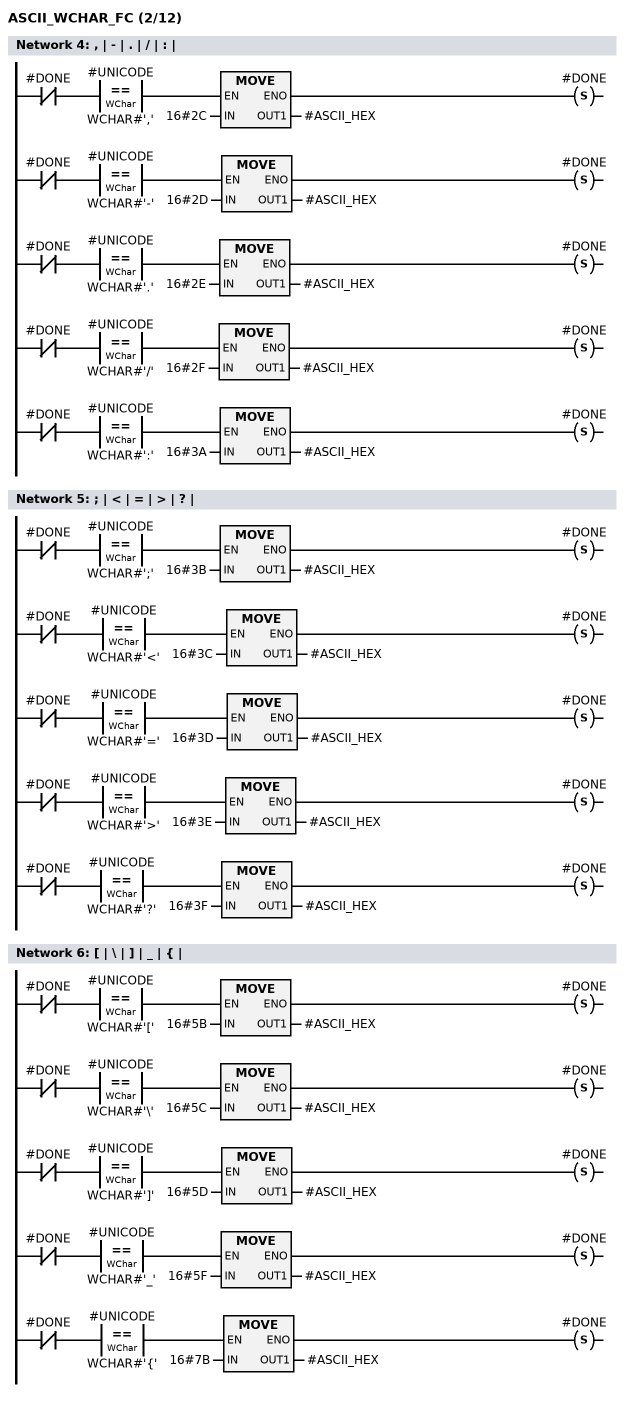
   RUNG wire#powerrail
      I_Contact( #DONE )
      { S7_Templates := "SrcType := WChar" } EQ_Contact(in1 := #UNICODE, in2 := WCHAR#',')
      Move(in := 16#2C, out1 => #ASCII_HEX)
      S_Coil( #DONE )
   END_RUNG
   RUNG wire#powerrail
      I_Contact( #DONE )
      { S7_Templates := "SrcType := WChar" } EQ_Contact(in1 := #UNICODE, in2 := WCHAR#'-')
      Move(in := 16#2D, out1 => #ASCII_HEX)
      S_Coil( #DONE )
   END_RUNG
   RUNG wire#powerrail
      I_Contact( #DONE )
      { S7_Templates := "SrcType := WChar" } EQ_Contact(in1 := #UNICODE, in2 := WCHAR#'.')
      Move(in := 16#2E, out1 => #ASCII_HEX)
      S_Coil( #DONE )
   END_RUNG
   RUNG wire#powerrail
      I_Contact( #DONE )
      { S7_Templates := "SrcType := WChar" } EQ_Contact(in1 := #UNICODE, in2 := WCHAR#'/')
      Move(in := 16#2F, out1 => #ASCII_HEX)
      S_Coil( #DONE )
   END_RUNG
   RUNG wire#powerrail
      I_Contact( #DONE )
      { S7_Templates := "SrcType := WChar" } EQ_Contact(in1 := #UNICODE, in2 := WCHAR#':')
      Move(in := 16#3A, out1 => #ASCII_HEX)
      S_Coil( #DONE )
   END_RUNG
   // the same network as SCL:
   IF NOT #DONE AND (#UNICODE = WCHAR#',') THEN
       #ASCII_HEX := 16#2C;
       #DONE := TRUE;
   END_IF;
   IF NOT #DONE AND (#UNICODE = WCHAR#'-') THEN
       #ASCII_HEX := 16#2D;
       #DONE := TRUE;
   END_IF;
   IF NOT #DONE AND (#UNICODE = WCHAR#'.') THEN
       #ASCII_HEX := 16#2E;
       #DONE := TRUE;
   END_IF;
   IF NOT #DONE AND (#UNICODE = WCHAR#'/') THEN
       #ASCII_HEX := 16#2F;
       #DONE := TRUE;
   END_IF;
   IF NOT #DONE AND (#UNICODE = WCHAR#':') THEN
       #ASCII_HEX := 16#3A;
       #DONE := TRUE;
   END_IF;
END_REGION

REGION Network 5: ; | < | = | > | ? |
   RUNG wire#powerrail
      I_Contact( #DONE )
      { S7_Templates := "SrcType := WChar" } EQ_Contact(in1 := #UNICODE, in2 := WCHAR#';')
      Move(in := 16#3B, out1 => #ASCII_HEX)
      S_Coil( #DONE )
   END_RUNG
   RUNG wire#powerrail
      I_Contact( #DONE )
      { S7_Templates := "SrcType := WChar" } EQ_Contact(in1 := #UNICODE, in2 := WCHAR#'<')
      Move(in := 16#3C, out1 => #ASCII_HEX)
      S_Coil( #DONE )
   END_RUNG
   RUNG wire#powerrail
      I_Contact( #DONE )
      { S7_Templates := "SrcType := WChar" } EQ_Contact(in1 := #UNICODE, in2 := WCHAR#'=')
      Move(in := 16#3D, out1 => #ASCII_HEX)
      S_Coil( #DONE )
   END_RUNG
   RUNG wire#powerrail
      I_Contact( #DONE )
      { S7_Templates := "SrcType := WChar" } EQ_Contact(in1 := #UNICODE, in2 := WCHAR#'>')
      Move(in := 16#3E, out1 => #ASCII_HEX)
      S_Coil( #DONE )
   END_RUNG
   RUNG wire#powerrail
      I_Contact( #DONE )
      { S7_Templates := "SrcType := WChar" } EQ_Contact(in1 := #UNICODE, in2 := WCHAR#'?')
      Move(in := 16#3F, out1 => #ASCII_HEX)
      S_Coil( #DONE )
   END_RUNG
   // the same network as SCL:
   IF NOT #DONE AND (#UNICODE = WCHAR#';') THEN
       #ASCII_HEX := 16#3B;
       #DONE := TRUE;
   END_IF;
   IF NOT #DONE AND (#UNICODE = WCHAR#'<') THEN
       #ASCII_HEX := 16#3C;
       #DONE := TRUE;
   END_IF;
   IF NOT #DONE AND (#UNICODE = WCHAR#'=') THEN
       #ASCII_HEX := 16#3D;
       #DONE := TRUE;
   END_IF;
   IF NOT #DONE AND (#UNICODE = WCHAR#'>') THEN
       #ASCII_HEX := 16#3E;
       #DONE := TRUE;
   END_IF;
   IF NOT #DONE AND (#UNICODE = WCHAR#'?') THEN
       #ASCII_HEX := 16#3F;
       #DONE := TRUE;
   END_IF;
END_REGION

REGION Network 6: [ | \ | ] | _ | { |
   RUNG wire#powerrail
      I_Contact( #DONE )
      { S7_Templates := "SrcType := WChar" } EQ_Contact(in1 := #UNICODE, in2 := WCHAR#'[')
      Move(in := 16#5B, out1 => #ASCII_HEX)
      S_Coil( #DONE )
   END_RUNG
   RUNG wire#powerrail
      I_Contact( #DONE )
      { S7_Templates := "SrcType := WChar" } EQ_Contact(in1 := #UNICODE, in2 := WCHAR#'\')
      Move(in := 16#5C, out1 => #ASCII_HEX)
      S_Coil( #DONE )
   END_RUNG
   RUNG wire#powerrail
      I_Contact( #DONE )
      { S7_Templates := "SrcType := WChar" } EQ_Contact(in1 := #UNICODE, in2 := WCHAR#']')
      Move(in := 16#5D, out1 => #ASCII_HEX)
      S_Coil( #DONE )
   END_RUNG
   RUNG wire#powerrail
      I_Contact( #DONE )
      { S7_Templates := "SrcType := WChar" } EQ_Contact(in1 := #UNICODE, in2 := WCHAR#'_')
      Move(in := 16#5F, out1 => #ASCII_HEX)
      S_Coil( #DONE )
   END_RUNG
   RUNG wire#powerrail
      I_Contact( #DONE )
      { S7_Templates := "SrcType := WChar" } EQ_Contact(in1 := #UNICODE, in2 := WCHAR#'{')
      Move(in := 16#7B, out1 => #ASCII_HEX)
      S_Coil( #DONE )
   END_RUNG
   // the same network as SCL:
   IF NOT #DONE AND (#UNICODE = WCHAR#'[') THEN
       #ASCII_HEX := 16#5B;
       #DONE := TRUE;
   END_IF;
   IF NOT #DONE AND (#UNICODE = WCHAR#'\') THEN
       #ASCII_HEX := 16#5C;
       #DONE := TRUE;
   END_IF;
   IF NOT #DONE AND (#UNICODE = WCHAR#']') THEN
       #ASCII_HEX := 16#5D;
       #DONE := TRUE;
   END_IF;
   IF NOT #DONE AND (#UNICODE = WCHAR#'_') THEN
       #ASCII_HEX := 16#5F;
       #DONE := TRUE;
   END_IF;
   IF NOT #DONE AND (#UNICODE = WCHAR#'{') THEN
       #ASCII_HEX := 16#7B;
       #DONE := TRUE;
   END_IF;
END_REGION

REGION Network 7: } | | |
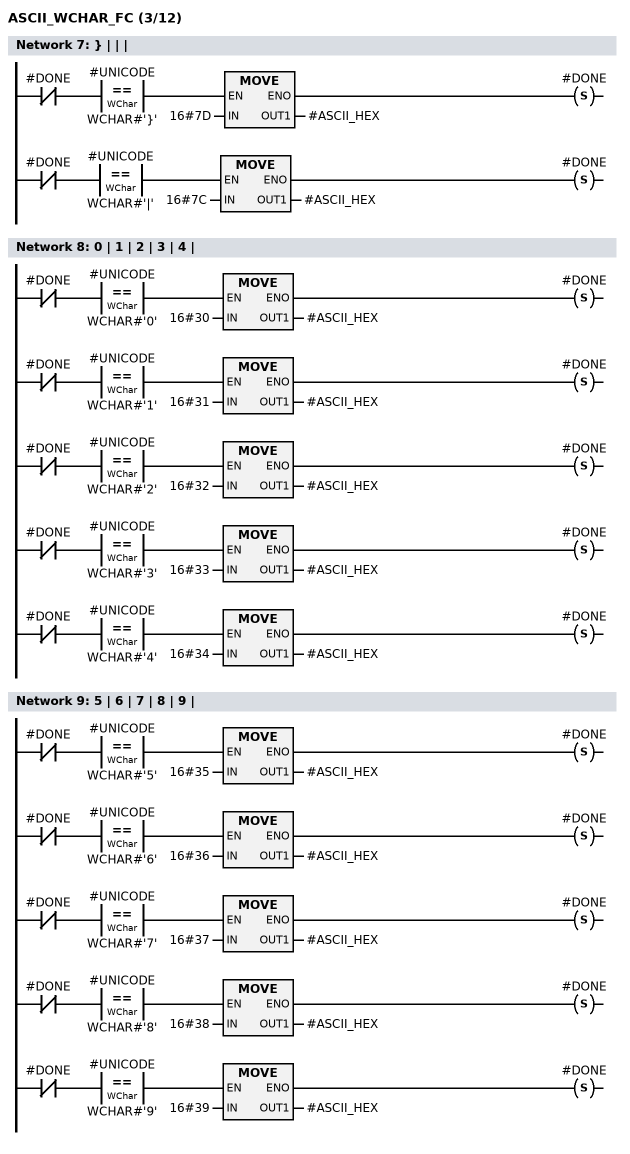
   RUNG wire#powerrail
      I_Contact( #DONE )
      { S7_Templates := "SrcType := WChar" } EQ_Contact(in1 := #UNICODE, in2 := WCHAR#'}')
      Move(in := 16#7D, out1 => #ASCII_HEX)
      S_Coil( #DONE )
   END_RUNG
   RUNG wire#powerrail
      I_Contact( #DONE )
      { S7_Templates := "SrcType := WChar" } EQ_Contact(in1 := #UNICODE, in2 := WCHAR#'|')
      Move(in := 16#7C, out1 => #ASCII_HEX)
      S_Coil( #DONE )
   END_RUNG
   // the same network as SCL:
   IF NOT #DONE AND (#UNICODE = WCHAR#'}') THEN
       #ASCII_HEX := 16#7D;
       #DONE := TRUE;
   END_IF;
   IF NOT #DONE AND (#UNICODE = WCHAR#'|') THEN
       #ASCII_HEX := 16#7C;
       #DONE := TRUE;
   END_IF;
END_REGION

REGION Network 8: 0 | 1 | 2 | 3 | 4 |
   RUNG wire#powerrail
      I_Contact( #DONE )
      { S7_Templates := "SrcType := WChar" } EQ_Contact(in1 := #UNICODE, in2 := WCHAR#'0')
      Move(in := 16#30, out1 => #ASCII_HEX)
      S_Coil( #DONE )
   END_RUNG
   RUNG wire#powerrail
      I_Contact( #DONE )
      { S7_Templates := "SrcType := WChar" } EQ_Contact(in1 := #UNICODE, in2 := WCHAR#'1')
      Move(in := 16#31, out1 => #ASCII_HEX)
      S_Coil( #DONE )
   END_RUNG
   RUNG wire#powerrail
      I_Contact( #DONE )
      { S7_Templates := "SrcType := WChar" } EQ_Contact(in1 := #UNICODE, in2 := WCHAR#'2')
      Move(in := 16#32, out1 => #ASCII_HEX)
      S_Coil( #DONE )
   END_RUNG
   RUNG wire#powerrail
      I_Contact( #DONE )
      { S7_Templates := "SrcType := WChar" } EQ_Contact(in1 := #UNICODE, in2 := WCHAR#'3')
      Move(in := 16#33, out1 => #ASCII_HEX)
      S_Coil( #DONE )
   END_RUNG
   RUNG wire#powerrail
      I_Contact( #DONE )
      { S7_Templates := "SrcType := WChar" } EQ_Contact(in1 := #UNICODE, in2 := WCHAR#'4')
      Move(in := 16#34, out1 => #ASCII_HEX)
      S_Coil( #DONE )
   END_RUNG
   // the same network as SCL:
   IF NOT #DONE AND (#UNICODE = WCHAR#'0') THEN
       #ASCII_HEX := 16#30;
       #DONE := TRUE;
   END_IF;
   IF NOT #DONE AND (#UNICODE = WCHAR#'1') THEN
       #ASCII_HEX := 16#31;
       #DONE := TRUE;
   END_IF;
   IF NOT #DONE AND (#UNICODE = WCHAR#'2') THEN
       #ASCII_HEX := 16#32;
       #DONE := TRUE;
   END_IF;
   IF NOT #DONE AND (#UNICODE = WCHAR#'3') THEN
       #ASCII_HEX := 16#33;
       #DONE := TRUE;
   END_IF;
   IF NOT #DONE AND (#UNICODE = WCHAR#'4') THEN
       #ASCII_HEX := 16#34;
       #DONE := TRUE;
   END_IF;
END_REGION

REGION Network 9: 5 | 6 | 7 | 8 | 9 |
   RUNG wire#powerrail
      I_Contact( #DONE )
      { S7_Templates := "SrcType := WChar" } EQ_Contact(in1 := #UNICODE, in2 := WCHAR#'5')
      Move(in := 16#35, out1 => #ASCII_HEX)
      S_Coil( #DONE )
   END_RUNG
   RUNG wire#powerrail
      I_Contact( #DONE )
      { S7_Templates := "SrcType := WChar" } EQ_Contact(in1 := #UNICODE, in2 := WCHAR#'6')
      Move(in := 16#36, out1 => #ASCII_HEX)
      S_Coil( #DONE )
   END_RUNG
   RUNG wire#powerrail
      I_Contact( #DONE )
      { S7_Templates := "SrcType := WChar" } EQ_Contact(in1 := #UNICODE, in2 := WCHAR#'7')
      Move(in := 16#37, out1 => #ASCII_HEX)
      S_Coil( #DONE )
   END_RUNG
   RUNG wire#powerrail
      I_Contact( #DONE )
      { S7_Templates := "SrcType := WChar" } EQ_Contact(in1 := #UNICODE, in2 := WCHAR#'8')
      Move(in := 16#38, out1 => #ASCII_HEX)
      S_Coil( #DONE )
   END_RUNG
   RUNG wire#powerrail
      I_Contact( #DONE )
      { S7_Templates := "SrcType := WChar" } EQ_Contact(in1 := #UNICODE, in2 := WCHAR#'9')
      Move(in := 16#39, out1 => #ASCII_HEX)
      S_Coil( #DONE )
   END_RUNG
   // the same network as SCL:
   IF NOT #DONE AND (#UNICODE = WCHAR#'5') THEN
       #ASCII_HEX := 16#35;
       #DONE := TRUE;
   END_IF;
   IF NOT #DONE AND (#UNICODE = WCHAR#'6') THEN
       #ASCII_HEX := 16#36;
       #DONE := TRUE;
   END_IF;
   IF NOT #DONE AND (#UNICODE = WCHAR#'7') THEN
       #ASCII_HEX := 16#37;
       #DONE := TRUE;
   END_IF;
   IF NOT #DONE AND (#UNICODE = WCHAR#'8') THEN
       #ASCII_HEX := 16#38;
       #DONE := TRUE;
   END_IF;
   IF NOT #DONE AND (#UNICODE = WCHAR#'9') THEN
       #ASCII_HEX := 16#39;
       #DONE := TRUE;
   END_IF;
END_REGION

REGION Network 10: А | Б | В | Г | Д |
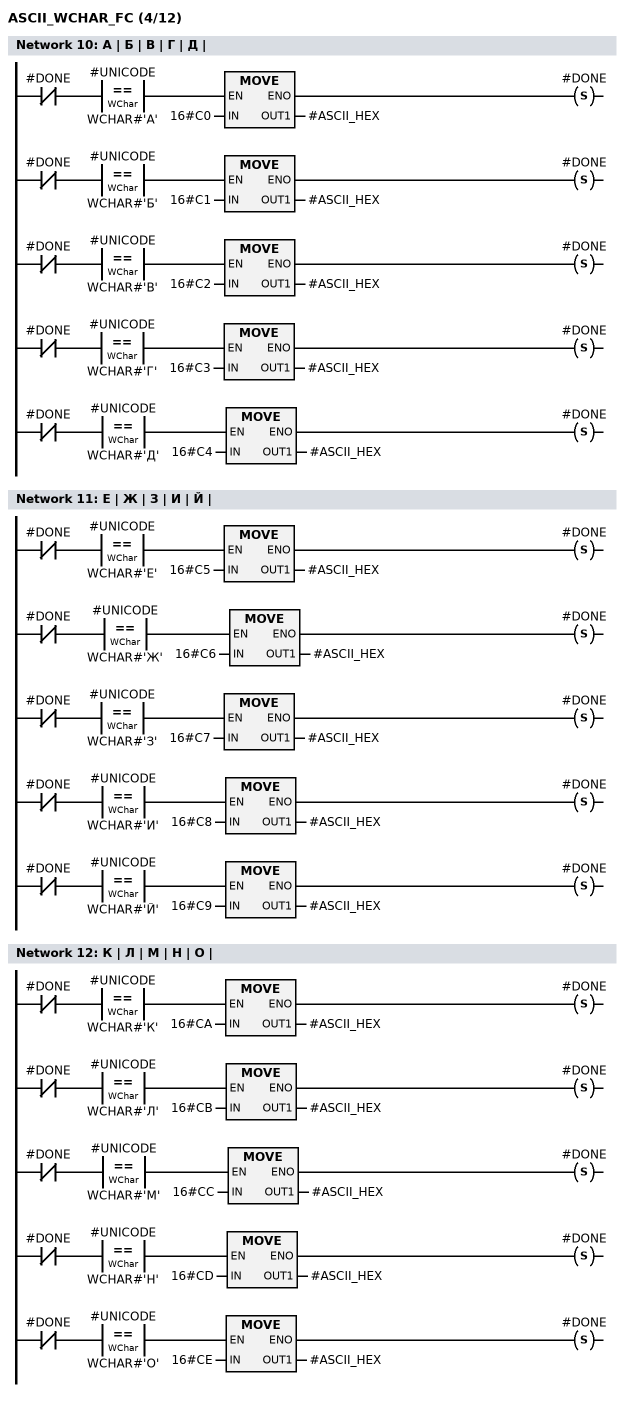
   RUNG wire#powerrail
      I_Contact( #DONE )
      { S7_Templates := "SrcType := WChar" } EQ_Contact(in1 := #UNICODE, in2 := WCHAR#'А')
      Move(in := 16#C0, out1 => #ASCII_HEX)
      S_Coil( #DONE )
   END_RUNG
   RUNG wire#powerrail
      I_Contact( #DONE )
      { S7_Templates := "SrcType := WChar" } EQ_Contact(in1 := #UNICODE, in2 := WCHAR#'Б')
      Move(in := 16#C1, out1 => #ASCII_HEX)
      S_Coil( #DONE )
   END_RUNG
   RUNG wire#powerrail
      I_Contact( #DONE )
      { S7_Templates := "SrcType := WChar" } EQ_Contact(in1 := #UNICODE, in2 := WCHAR#'В')
      Move(in := 16#C2, out1 => #ASCII_HEX)
      S_Coil( #DONE )
   END_RUNG
   RUNG wire#powerrail
      I_Contact( #DONE )
      { S7_Templates := "SrcType := WChar" } EQ_Contact(in1 := #UNICODE, in2 := WCHAR#'Г')
      Move(in := 16#C3, out1 => #ASCII_HEX)
      S_Coil( #DONE )
   END_RUNG
   RUNG wire#powerrail
      I_Contact( #DONE )
      { S7_Templates := "SrcType := WChar" } EQ_Contact(in1 := #UNICODE, in2 := WCHAR#'Д')
      Move(in := 16#C4, out1 => #ASCII_HEX)
      S_Coil( #DONE )
   END_RUNG
   // the same network as SCL:
   IF NOT #DONE AND (#UNICODE = WCHAR#'А') THEN
       #ASCII_HEX := 16#C0;
       #DONE := TRUE;
   END_IF;
   IF NOT #DONE AND (#UNICODE = WCHAR#'Б') THEN
       #ASCII_HEX := 16#C1;
       #DONE := TRUE;
   END_IF;
   IF NOT #DONE AND (#UNICODE = WCHAR#'В') THEN
       #ASCII_HEX := 16#C2;
       #DONE := TRUE;
   END_IF;
   IF NOT #DONE AND (#UNICODE = WCHAR#'Г') THEN
       #ASCII_HEX := 16#C3;
       #DONE := TRUE;
   END_IF;
   IF NOT #DONE AND (#UNICODE = WCHAR#'Д') THEN
       #ASCII_HEX := 16#C4;
       #DONE := TRUE;
   END_IF;
END_REGION

REGION Network 11: Е | Ж | З | И | Й |
   RUNG wire#powerrail
      I_Contact( #DONE )
      { S7_Templates := "SrcType := WChar" } EQ_Contact(in1 := #UNICODE, in2 := WCHAR#'Е')
      Move(in := 16#C5, out1 => #ASCII_HEX)
      S_Coil( #DONE )
   END_RUNG
   RUNG wire#powerrail
      I_Contact( #DONE )
      { S7_Templates := "SrcType := WChar" } EQ_Contact(in1 := #UNICODE, in2 := WCHAR#'Ж')
      Move(in := 16#C6, out1 => #ASCII_HEX)
      S_Coil( #DONE )
   END_RUNG
   RUNG wire#powerrail
      I_Contact( #DONE )
      { S7_Templates := "SrcType := WChar" } EQ_Contact(in1 := #UNICODE, in2 := WCHAR#'З')
      Move(in := 16#C7, out1 => #ASCII_HEX)
      S_Coil( #DONE )
   END_RUNG
   RUNG wire#powerrail
      I_Contact( #DONE )
      { S7_Templates := "SrcType := WChar" } EQ_Contact(in1 := #UNICODE, in2 := WCHAR#'И')
      Move(in := 16#C8, out1 => #ASCII_HEX)
      S_Coil( #DONE )
   END_RUNG
   RUNG wire#powerrail
      I_Contact( #DONE )
      { S7_Templates := "SrcType := WChar" } EQ_Contact(in1 := #UNICODE, in2 := WCHAR#'Й')
      Move(in := 16#C9, out1 => #ASCII_HEX)
      S_Coil( #DONE )
   END_RUNG
   // the same network as SCL:
   IF NOT #DONE AND (#UNICODE = WCHAR#'Е') THEN
       #ASCII_HEX := 16#C5;
       #DONE := TRUE;
   END_IF;
   IF NOT #DONE AND (#UNICODE = WCHAR#'Ж') THEN
       #ASCII_HEX := 16#C6;
       #DONE := TRUE;
   END_IF;
   IF NOT #DONE AND (#UNICODE = WCHAR#'З') THEN
       #ASCII_HEX := 16#C7;
       #DONE := TRUE;
   END_IF;
   IF NOT #DONE AND (#UNICODE = WCHAR#'И') THEN
       #ASCII_HEX := 16#C8;
       #DONE := TRUE;
   END_IF;
   IF NOT #DONE AND (#UNICODE = WCHAR#'Й') THEN
       #ASCII_HEX := 16#C9;
       #DONE := TRUE;
   END_IF;
END_REGION

REGION Network 12: К | Л | М | Н | О |
   RUNG wire#powerrail
      I_Contact( #DONE )
      { S7_Templates := "SrcType := WChar" } EQ_Contact(in1 := #UNICODE, in2 := WCHAR#'К')
      Move(in := 16#CA, out1 => #ASCII_HEX)
      S_Coil( #DONE )
   END_RUNG
   RUNG wire#powerrail
      I_Contact( #DONE )
      { S7_Templates := "SrcType := WChar" } EQ_Contact(in1 := #UNICODE, in2 := WCHAR#'Л')
      Move(in := 16#CB, out1 => #ASCII_HEX)
      S_Coil( #DONE )
   END_RUNG
   RUNG wire#powerrail
      I_Contact( #DONE )
      { S7_Templates := "SrcType := WChar" } EQ_Contact(in1 := #UNICODE, in2 := WCHAR#'М')
      Move(in := 16#CC, out1 => #ASCII_HEX)
      S_Coil( #DONE )
   END_RUNG
   RUNG wire#powerrail
      I_Contact( #DONE )
      { S7_Templates := "SrcType := WChar" } EQ_Contact(in1 := #UNICODE, in2 := WCHAR#'Н')
      Move(in := 16#CD, out1 => #ASCII_HEX)
      S_Coil( #DONE )
   END_RUNG
   RUNG wire#powerrail
      I_Contact( #DONE )
      { S7_Templates := "SrcType := WChar" } EQ_Contact(in1 := #UNICODE, in2 := WCHAR#'О')
      Move(in := 16#CE, out1 => #ASCII_HEX)
      S_Coil( #DONE )
   END_RUNG
   // the same network as SCL:
   IF NOT #DONE AND (#UNICODE = WCHAR#'К') THEN
       #ASCII_HEX := 16#CA;
       #DONE := TRUE;
   END_IF;
   IF NOT #DONE AND (#UNICODE = WCHAR#'Л') THEN
       #ASCII_HEX := 16#CB;
       #DONE := TRUE;
   END_IF;
   IF NOT #DONE AND (#UNICODE = WCHAR#'М') THEN
       #ASCII_HEX := 16#CC;
       #DONE := TRUE;
   END_IF;
   IF NOT #DONE AND (#UNICODE = WCHAR#'Н') THEN
       #ASCII_HEX := 16#CD;
       #DONE := TRUE;
   END_IF;
   IF NOT #DONE AND (#UNICODE = WCHAR#'О') THEN
       #ASCII_HEX := 16#CE;
       #DONE := TRUE;
   END_IF;
END_REGION

REGION Network 13: П | Р | С | Т | У |
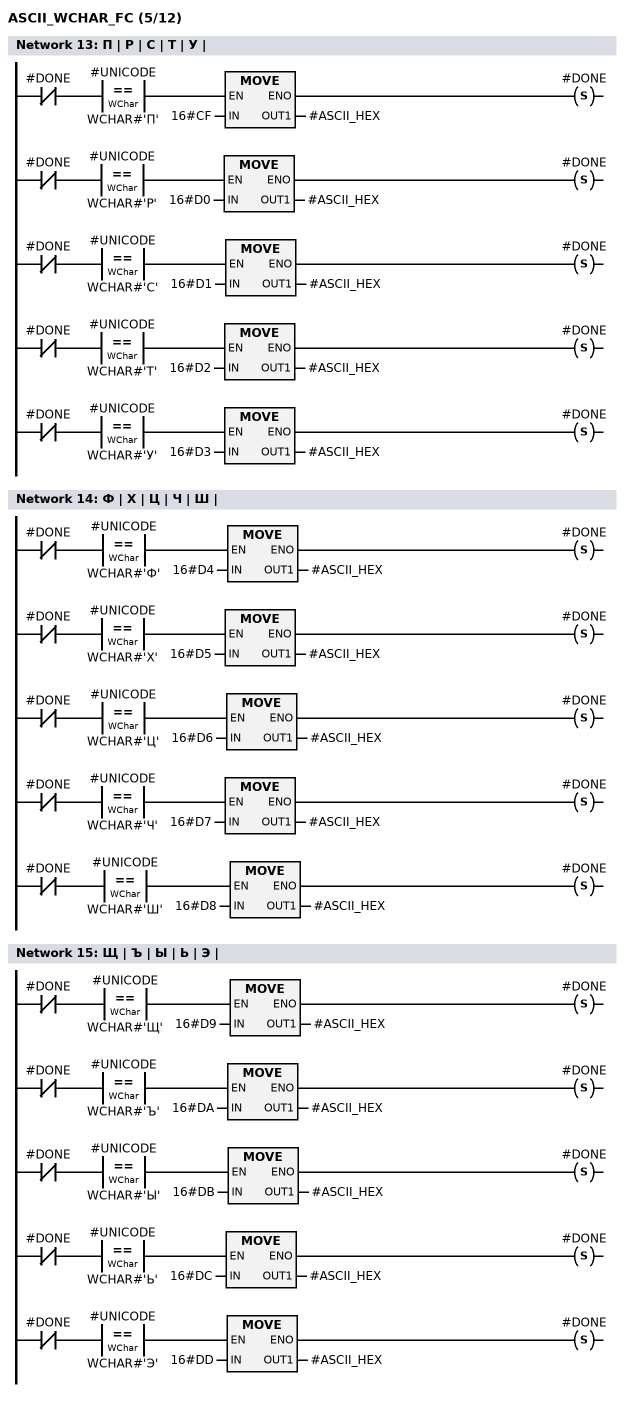
   RUNG wire#powerrail
      I_Contact( #DONE )
      { S7_Templates := "SrcType := WChar" } EQ_Contact(in1 := #UNICODE, in2 := WCHAR#'П')
      Move(in := 16#CF, out1 => #ASCII_HEX)
      S_Coil( #DONE )
   END_RUNG
   RUNG wire#powerrail
      I_Contact( #DONE )
      { S7_Templates := "SrcType := WChar" } EQ_Contact(in1 := #UNICODE, in2 := WCHAR#'Р')
      Move(in := 16#D0, out1 => #ASCII_HEX)
      S_Coil( #DONE )
   END_RUNG
   RUNG wire#powerrail
      I_Contact( #DONE )
      { S7_Templates := "SrcType := WChar" } EQ_Contact(in1 := #UNICODE, in2 := WCHAR#'С')
      Move(in := 16#D1, out1 => #ASCII_HEX)
      S_Coil( #DONE )
   END_RUNG
   RUNG wire#powerrail
      I_Contact( #DONE )
      { S7_Templates := "SrcType := WChar" } EQ_Contact(in1 := #UNICODE, in2 := WCHAR#'Т')
      Move(in := 16#D2, out1 => #ASCII_HEX)
      S_Coil( #DONE )
   END_RUNG
   RUNG wire#powerrail
      I_Contact( #DONE )
      { S7_Templates := "SrcType := WChar" } EQ_Contact(in1 := #UNICODE, in2 := WCHAR#'У')
      Move(in := 16#D3, out1 => #ASCII_HEX)
      S_Coil( #DONE )
   END_RUNG
   // the same network as SCL:
   IF NOT #DONE AND (#UNICODE = WCHAR#'П') THEN
       #ASCII_HEX := 16#CF;
       #DONE := TRUE;
   END_IF;
   IF NOT #DONE AND (#UNICODE = WCHAR#'Р') THEN
       #ASCII_HEX := 16#D0;
       #DONE := TRUE;
   END_IF;
   IF NOT #DONE AND (#UNICODE = WCHAR#'С') THEN
       #ASCII_HEX := 16#D1;
       #DONE := TRUE;
   END_IF;
   IF NOT #DONE AND (#UNICODE = WCHAR#'Т') THEN
       #ASCII_HEX := 16#D2;
       #DONE := TRUE;
   END_IF;
   IF NOT #DONE AND (#UNICODE = WCHAR#'У') THEN
       #ASCII_HEX := 16#D3;
       #DONE := TRUE;
   END_IF;
END_REGION

REGION Network 14: Ф | Х | Ц | Ч | Ш |
   RUNG wire#powerrail
      I_Contact( #DONE )
      { S7_Templates := "SrcType := WChar" } EQ_Contact(in1 := #UNICODE, in2 := WCHAR#'Ф')
      Move(in := 16#D4, out1 => #ASCII_HEX)
      S_Coil( #DONE )
   END_RUNG
   RUNG wire#powerrail
      I_Contact( #DONE )
      { S7_Templates := "SrcType := WChar" } EQ_Contact(in1 := #UNICODE, in2 := WCHAR#'Х')
      Move(in := 16#D5, out1 => #ASCII_HEX)
      S_Coil( #DONE )
   END_RUNG
   RUNG wire#powerrail
      I_Contact( #DONE )
      { S7_Templates := "SrcType := WChar" } EQ_Contact(in1 := #UNICODE, in2 := WCHAR#'Ц')
      Move(in := 16#D6, out1 => #ASCII_HEX)
      S_Coil( #DONE )
   END_RUNG
   RUNG wire#powerrail
      I_Contact( #DONE )
      { S7_Templates := "SrcType := WChar" } EQ_Contact(in1 := #UNICODE, in2 := WCHAR#'Ч')
      Move(in := 16#D7, out1 => #ASCII_HEX)
      S_Coil( #DONE )
   END_RUNG
   RUNG wire#powerrail
      I_Contact( #DONE )
      { S7_Templates := "SrcType := WChar" } EQ_Contact(in1 := #UNICODE, in2 := WCHAR#'Ш')
      Move(in := 16#D8, out1 => #ASCII_HEX)
      S_Coil( #DONE )
   END_RUNG
   // the same network as SCL:
   IF NOT #DONE AND (#UNICODE = WCHAR#'Ф') THEN
       #ASCII_HEX := 16#D4;
       #DONE := TRUE;
   END_IF;
   IF NOT #DONE AND (#UNICODE = WCHAR#'Х') THEN
       #ASCII_HEX := 16#D5;
       #DONE := TRUE;
   END_IF;
   IF NOT #DONE AND (#UNICODE = WCHAR#'Ц') THEN
       #ASCII_HEX := 16#D6;
       #DONE := TRUE;
   END_IF;
   IF NOT #DONE AND (#UNICODE = WCHAR#'Ч') THEN
       #ASCII_HEX := 16#D7;
       #DONE := TRUE;
   END_IF;
   IF NOT #DONE AND (#UNICODE = WCHAR#'Ш') THEN
       #ASCII_HEX := 16#D8;
       #DONE := TRUE;
   END_IF;
END_REGION

REGION Network 15: Щ | Ъ | Ы | Ь | Э |
   RUNG wire#powerrail
      I_Contact( #DONE )
      { S7_Templates := "SrcType := WChar" } EQ_Contact(in1 := #UNICODE, in2 := WCHAR#'Щ')
      Move(in := 16#D9, out1 => #ASCII_HEX)
      S_Coil( #DONE )
   END_RUNG
   RUNG wire#powerrail
      I_Contact( #DONE )
      { S7_Templates := "SrcType := WChar" } EQ_Contact(in1 := #UNICODE, in2 := WCHAR#'Ъ')
      Move(in := 16#DA, out1 => #ASCII_HEX)
      S_Coil( #DONE )
   END_RUNG
   RUNG wire#powerrail
      I_Contact( #DONE )
      { S7_Templates := "SrcType := WChar" } EQ_Contact(in1 := #UNICODE, in2 := WCHAR#'Ы')
      Move(in := 16#DB, out1 => #ASCII_HEX)
      S_Coil( #DONE )
   END_RUNG
   RUNG wire#powerrail
      I_Contact( #DONE )
      { S7_Templates := "SrcType := WChar" } EQ_Contact(in1 := #UNICODE, in2 := WCHAR#'Ь')
      Move(in := 16#DC, out1 => #ASCII_HEX)
      S_Coil( #DONE )
   END_RUNG
   RUNG wire#powerrail
      I_Contact( #DONE )
      { S7_Templates := "SrcType := WChar" } EQ_Contact(in1 := #UNICODE, in2 := WCHAR#'Э')
      Move(in := 16#DD, out1 => #ASCII_HEX)
      S_Coil( #DONE )
   END_RUNG
   // the same network as SCL:
   IF NOT #DONE AND (#UNICODE = WCHAR#'Щ') THEN
       #ASCII_HEX := 16#D9;
       #DONE := TRUE;
   END_IF;
   IF NOT #DONE AND (#UNICODE = WCHAR#'Ъ') THEN
       #ASCII_HEX := 16#DA;
       #DONE := TRUE;
   END_IF;
   IF NOT #DONE AND (#UNICODE = WCHAR#'Ы') THEN
       #ASCII_HEX := 16#DB;
       #DONE := TRUE;
   END_IF;
   IF NOT #DONE AND (#UNICODE = WCHAR#'Ь') THEN
       #ASCII_HEX := 16#DC;
       #DONE := TRUE;
   END_IF;
   IF NOT #DONE AND (#UNICODE = WCHAR#'Э') THEN
       #ASCII_HEX := 16#DD;
       #DONE := TRUE;
   END_IF;
END_REGION

REGION Network 16: Ю | Я |
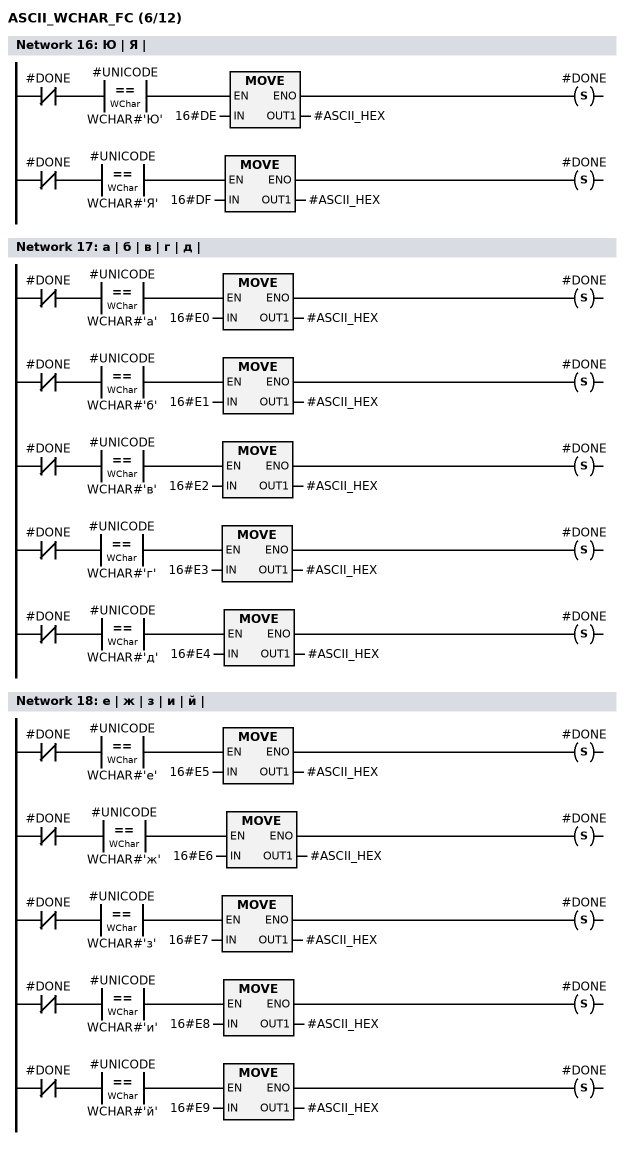
   RUNG wire#powerrail
      I_Contact( #DONE )
      { S7_Templates := "SrcType := WChar" } EQ_Contact(in1 := #UNICODE, in2 := WCHAR#'Ю')
      Move(in := 16#DE, out1 => #ASCII_HEX)
      S_Coil( #DONE )
   END_RUNG
   RUNG wire#powerrail
      I_Contact( #DONE )
      { S7_Templates := "SrcType := WChar" } EQ_Contact(in1 := #UNICODE, in2 := WCHAR#'Я')
      Move(in := 16#DF, out1 => #ASCII_HEX)
      S_Coil( #DONE )
   END_RUNG
   // the same network as SCL:
   IF NOT #DONE AND (#UNICODE = WCHAR#'Ю') THEN
       #ASCII_HEX := 16#DE;
       #DONE := TRUE;
   END_IF;
   IF NOT #DONE AND (#UNICODE = WCHAR#'Я') THEN
       #ASCII_HEX := 16#DF;
       #DONE := TRUE;
   END_IF;
END_REGION

REGION Network 17: а | б | в | г | д |
   RUNG wire#powerrail
      I_Contact( #DONE )
      { S7_Templates := "SrcType := WChar" } EQ_Contact(in1 := #UNICODE, in2 := WCHAR#'а')
      Move(in := 16#E0, out1 => #ASCII_HEX)
      S_Coil( #DONE )
   END_RUNG
   RUNG wire#powerrail
      I_Contact( #DONE )
      { S7_Templates := "SrcType := WChar" } EQ_Contact(in1 := #UNICODE, in2 := WCHAR#'б')
      Move(in := 16#E1, out1 => #ASCII_HEX)
      S_Coil( #DONE )
   END_RUNG
   RUNG wire#powerrail
      I_Contact( #DONE )
      { S7_Templates := "SrcType := WChar" } EQ_Contact(in1 := #UNICODE, in2 := WCHAR#'в')
      Move(in := 16#E2, out1 => #ASCII_HEX)
      S_Coil( #DONE )
   END_RUNG
   RUNG wire#powerrail
      I_Contact( #DONE )
      { S7_Templates := "SrcType := WChar" } EQ_Contact(in1 := #UNICODE, in2 := WCHAR#'г')
      Move(in := 16#E3, out1 => #ASCII_HEX)
      S_Coil( #DONE )
   END_RUNG
   RUNG wire#powerrail
      I_Contact( #DONE )
      { S7_Templates := "SrcType := WChar" } EQ_Contact(in1 := #UNICODE, in2 := WCHAR#'д')
      Move(in := 16#E4, out1 => #ASCII_HEX)
      S_Coil( #DONE )
   END_RUNG
   // the same network as SCL:
   IF NOT #DONE AND (#UNICODE = WCHAR#'а') THEN
       #ASCII_HEX := 16#E0;
       #DONE := TRUE;
   END_IF;
   IF NOT #DONE AND (#UNICODE = WCHAR#'б') THEN
       #ASCII_HEX := 16#E1;
       #DONE := TRUE;
   END_IF;
   IF NOT #DONE AND (#UNICODE = WCHAR#'в') THEN
       #ASCII_HEX := 16#E2;
       #DONE := TRUE;
   END_IF;
   IF NOT #DONE AND (#UNICODE = WCHAR#'г') THEN
       #ASCII_HEX := 16#E3;
       #DONE := TRUE;
   END_IF;
   IF NOT #DONE AND (#UNICODE = WCHAR#'д') THEN
       #ASCII_HEX := 16#E4;
       #DONE := TRUE;
   END_IF;
END_REGION

REGION Network 18: е | ж | з | и | й |
   RUNG wire#powerrail
      I_Contact( #DONE )
      { S7_Templates := "SrcType := WChar" } EQ_Contact(in1 := #UNICODE, in2 := WCHAR#'е')
      Move(in := 16#E5, out1 => #ASCII_HEX)
      S_Coil( #DONE )
   END_RUNG
   RUNG wire#powerrail
      I_Contact( #DONE )
      { S7_Templates := "SrcType := WChar" } EQ_Contact(in1 := #UNICODE, in2 := WCHAR#'ж')
      Move(in := 16#E6, out1 => #ASCII_HEX)
      S_Coil( #DONE )
   END_RUNG
   RUNG wire#powerrail
      I_Contact( #DONE )
      { S7_Templates := "SrcType := WChar" } EQ_Contact(in1 := #UNICODE, in2 := WCHAR#'з')
      Move(in := 16#E7, out1 => #ASCII_HEX)
      S_Coil( #DONE )
   END_RUNG
   RUNG wire#powerrail
      I_Contact( #DONE )
      { S7_Templates := "SrcType := WChar" } EQ_Contact(in1 := #UNICODE, in2 := WCHAR#'и')
      Move(in := 16#E8, out1 => #ASCII_HEX)
      S_Coil( #DONE )
   END_RUNG
   RUNG wire#powerrail
      I_Contact( #DONE )
      { S7_Templates := "SrcType := WChar" } EQ_Contact(in1 := #UNICODE, in2 := WCHAR#'й')
      Move(in := 16#E9, out1 => #ASCII_HEX)
      S_Coil( #DONE )
   END_RUNG
   // the same network as SCL:
   IF NOT #DONE AND (#UNICODE = WCHAR#'е') THEN
       #ASCII_HEX := 16#E5;
       #DONE := TRUE;
   END_IF;
   IF NOT #DONE AND (#UNICODE = WCHAR#'ж') THEN
       #ASCII_HEX := 16#E6;
       #DONE := TRUE;
   END_IF;
   IF NOT #DONE AND (#UNICODE = WCHAR#'з') THEN
       #ASCII_HEX := 16#E7;
       #DONE := TRUE;
   END_IF;
   IF NOT #DONE AND (#UNICODE = WCHAR#'и') THEN
       #ASCII_HEX := 16#E8;
       #DONE := TRUE;
   END_IF;
   IF NOT #DONE AND (#UNICODE = WCHAR#'й') THEN
       #ASCII_HEX := 16#E9;
       #DONE := TRUE;
   END_IF;
END_REGION

REGION Network 19: к | л | м | н | о |
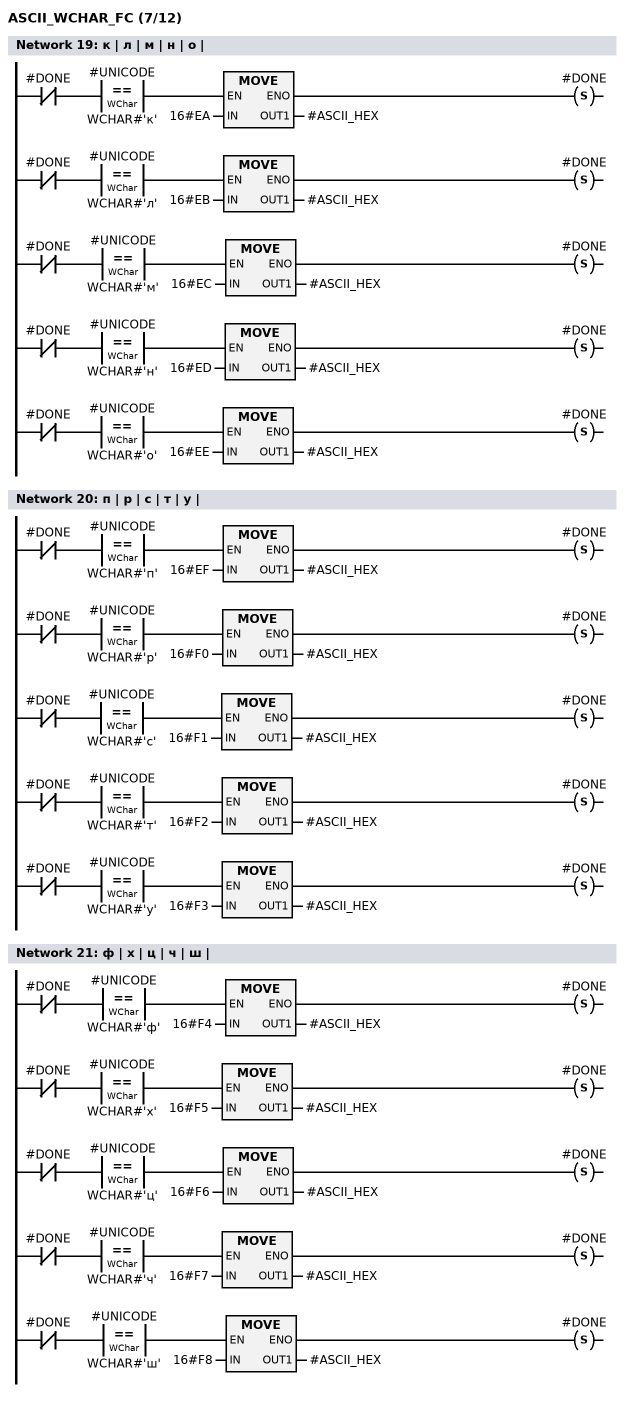
   RUNG wire#powerrail
      I_Contact( #DONE )
      { S7_Templates := "SrcType := WChar" } EQ_Contact(in1 := #UNICODE, in2 := WCHAR#'к')
      Move(in := 16#EA, out1 => #ASCII_HEX)
      S_Coil( #DONE )
   END_RUNG
   RUNG wire#powerrail
      I_Contact( #DONE )
      { S7_Templates := "SrcType := WChar" } EQ_Contact(in1 := #UNICODE, in2 := WCHAR#'л')
      Move(in := 16#EB, out1 => #ASCII_HEX)
      S_Coil( #DONE )
   END_RUNG
   RUNG wire#powerrail
      I_Contact( #DONE )
      { S7_Templates := "SrcType := WChar" } EQ_Contact(in1 := #UNICODE, in2 := WCHAR#'м')
      Move(in := 16#EC, out1 => #ASCII_HEX)
      S_Coil( #DONE )
   END_RUNG
   RUNG wire#powerrail
      I_Contact( #DONE )
      { S7_Templates := "SrcType := WChar" } EQ_Contact(in1 := #UNICODE, in2 := WCHAR#'н')
      Move(in := 16#ED, out1 => #ASCII_HEX)
      S_Coil( #DONE )
   END_RUNG
   RUNG wire#powerrail
      I_Contact( #DONE )
      { S7_Templates := "SrcType := WChar" } EQ_Contact(in1 := #UNICODE, in2 := WCHAR#'о')
      Move(in := 16#EE, out1 => #ASCII_HEX)
      S_Coil( #DONE )
   END_RUNG
   // the same network as SCL:
   IF NOT #DONE AND (#UNICODE = WCHAR#'к') THEN
       #ASCII_HEX := 16#EA;
       #DONE := TRUE;
   END_IF;
   IF NOT #DONE AND (#UNICODE = WCHAR#'л') THEN
       #ASCII_HEX := 16#EB;
       #DONE := TRUE;
   END_IF;
   IF NOT #DONE AND (#UNICODE = WCHAR#'м') THEN
       #ASCII_HEX := 16#EC;
       #DONE := TRUE;
   END_IF;
   IF NOT #DONE AND (#UNICODE = WCHAR#'н') THEN
       #ASCII_HEX := 16#ED;
       #DONE := TRUE;
   END_IF;
   IF NOT #DONE AND (#UNICODE = WCHAR#'о') THEN
       #ASCII_HEX := 16#EE;
       #DONE := TRUE;
   END_IF;
END_REGION

REGION Network 20: п | р | с | т | у |
   RUNG wire#powerrail
      I_Contact( #DONE )
      { S7_Templates := "SrcType := WChar" } EQ_Contact(in1 := #UNICODE, in2 := WCHAR#'п')
      Move(in := 16#EF, out1 => #ASCII_HEX)
      S_Coil( #DONE )
   END_RUNG
   RUNG wire#powerrail
      I_Contact( #DONE )
      { S7_Templates := "SrcType := WChar" } EQ_Contact(in1 := #UNICODE, in2 := WCHAR#'р')
      Move(in := 16#F0, out1 => #ASCII_HEX)
      S_Coil( #DONE )
   END_RUNG
   RUNG wire#powerrail
      I_Contact( #DONE )
      { S7_Templates := "SrcType := WChar" } EQ_Contact(in1 := #UNICODE, in2 := WCHAR#'с')
      Move(in := 16#F1, out1 => #ASCII_HEX)
      S_Coil( #DONE )
   END_RUNG
   RUNG wire#powerrail
      I_Contact( #DONE )
      { S7_Templates := "SrcType := WChar" } EQ_Contact(in1 := #UNICODE, in2 := WCHAR#'т')
      Move(in := 16#F2, out1 => #ASCII_HEX)
      S_Coil( #DONE )
   END_RUNG
   RUNG wire#powerrail
      I_Contact( #DONE )
      { S7_Templates := "SrcType := WChar" } EQ_Contact(in1 := #UNICODE, in2 := WCHAR#'у')
      Move(in := 16#F3, out1 => #ASCII_HEX)
      S_Coil( #DONE )
   END_RUNG
   // the same network as SCL:
   IF NOT #DONE AND (#UNICODE = WCHAR#'п') THEN
       #ASCII_HEX := 16#EF;
       #DONE := TRUE;
   END_IF;
   IF NOT #DONE AND (#UNICODE = WCHAR#'р') THEN
       #ASCII_HEX := 16#F0;
       #DONE := TRUE;
   END_IF;
   IF NOT #DONE AND (#UNICODE = WCHAR#'с') THEN
       #ASCII_HEX := 16#F1;
       #DONE := TRUE;
   END_IF;
   IF NOT #DONE AND (#UNICODE = WCHAR#'т') THEN
       #ASCII_HEX := 16#F2;
       #DONE := TRUE;
   END_IF;
   IF NOT #DONE AND (#UNICODE = WCHAR#'у') THEN
       #ASCII_HEX := 16#F3;
       #DONE := TRUE;
   END_IF;
END_REGION

REGION Network 21: ф | х | ц | ч | ш |
   RUNG wire#powerrail
      I_Contact( #DONE )
      { S7_Templates := "SrcType := WChar" } EQ_Contact(in1 := #UNICODE, in2 := WCHAR#'ф')
      Move(in := 16#F4, out1 => #ASCII_HEX)
      S_Coil( #DONE )
   END_RUNG
   RUNG wire#powerrail
      I_Contact( #DONE )
      { S7_Templates := "SrcType := WChar" } EQ_Contact(in1 := #UNICODE, in2 := WCHAR#'х')
      Move(in := 16#F5, out1 => #ASCII_HEX)
      S_Coil( #DONE )
   END_RUNG
   RUNG wire#powerrail
      I_Contact( #DONE )
      { S7_Templates := "SrcType := WChar" } EQ_Contact(in1 := #UNICODE, in2 := WCHAR#'ц')
      Move(in := 16#F6, out1 => #ASCII_HEX)
      S_Coil( #DONE )
   END_RUNG
   RUNG wire#powerrail
      I_Contact( #DONE )
      { S7_Templates := "SrcType := WChar" } EQ_Contact(in1 := #UNICODE, in2 := WCHAR#'ч')
      Move(in := 16#F7, out1 => #ASCII_HEX)
      S_Coil( #DONE )
   END_RUNG
   RUNG wire#powerrail
      I_Contact( #DONE )
      { S7_Templates := "SrcType := WChar" } EQ_Contact(in1 := #UNICODE, in2 := WCHAR#'ш')
      Move(in := 16#F8, out1 => #ASCII_HEX)
      S_Coil( #DONE )
   END_RUNG
   // the same network as SCL:
   IF NOT #DONE AND (#UNICODE = WCHAR#'ф') THEN
       #ASCII_HEX := 16#F4;
       #DONE := TRUE;
   END_IF;
   IF NOT #DONE AND (#UNICODE = WCHAR#'х') THEN
       #ASCII_HEX := 16#F5;
       #DONE := TRUE;
   END_IF;
   IF NOT #DONE AND (#UNICODE = WCHAR#'ц') THEN
       #ASCII_HEX := 16#F6;
       #DONE := TRUE;
   END_IF;
   IF NOT #DONE AND (#UNICODE = WCHAR#'ч') THEN
       #ASCII_HEX := 16#F7;
       #DONE := TRUE;
   END_IF;
   IF NOT #DONE AND (#UNICODE = WCHAR#'ш') THEN
       #ASCII_HEX := 16#F8;
       #DONE := TRUE;
   END_IF;
END_REGION

REGION Network 22: щ | ъ | ы | ь | э |
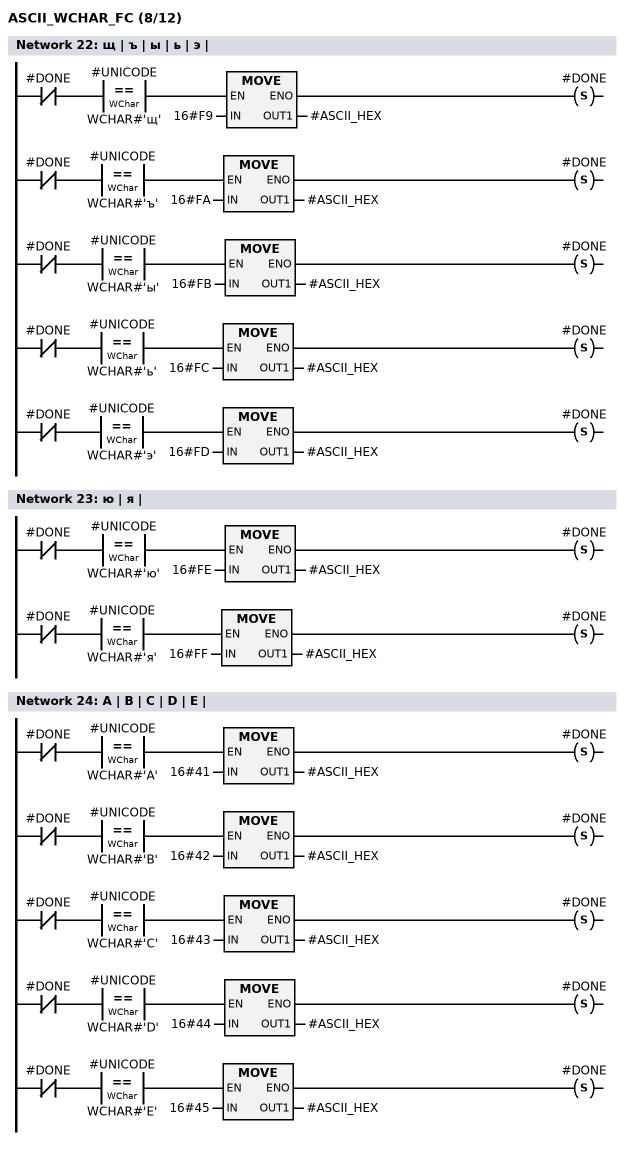
   RUNG wire#powerrail
      I_Contact( #DONE )
      { S7_Templates := "SrcType := WChar" } EQ_Contact(in1 := #UNICODE, in2 := WCHAR#'щ')
      Move(in := 16#F9, out1 => #ASCII_HEX)
      S_Coil( #DONE )
   END_RUNG
   RUNG wire#powerrail
      I_Contact( #DONE )
      { S7_Templates := "SrcType := WChar" } EQ_Contact(in1 := #UNICODE, in2 := WCHAR#'ъ')
      Move(in := 16#FA, out1 => #ASCII_HEX)
      S_Coil( #DONE )
   END_RUNG
   RUNG wire#powerrail
      I_Contact( #DONE )
      { S7_Templates := "SrcType := WChar" } EQ_Contact(in1 := #UNICODE, in2 := WCHAR#'ы')
      Move(in := 16#FB, out1 => #ASCII_HEX)
      S_Coil( #DONE )
   END_RUNG
   RUNG wire#powerrail
      I_Contact( #DONE )
      { S7_Templates := "SrcType := WChar" } EQ_Contact(in1 := #UNICODE, in2 := WCHAR#'ь')
      Move(in := 16#FC, out1 => #ASCII_HEX)
      S_Coil( #DONE )
   END_RUNG
   RUNG wire#powerrail
      I_Contact( #DONE )
      { S7_Templates := "SrcType := WChar" } EQ_Contact(in1 := #UNICODE, in2 := WCHAR#'э')
      Move(in := 16#FD, out1 => #ASCII_HEX)
      S_Coil( #DONE )
   END_RUNG
   // the same network as SCL:
   IF NOT #DONE AND (#UNICODE = WCHAR#'щ') THEN
       #ASCII_HEX := 16#F9;
       #DONE := TRUE;
   END_IF;
   IF NOT #DONE AND (#UNICODE = WCHAR#'ъ') THEN
       #ASCII_HEX := 16#FA;
       #DONE := TRUE;
   END_IF;
   IF NOT #DONE AND (#UNICODE = WCHAR#'ы') THEN
       #ASCII_HEX := 16#FB;
       #DONE := TRUE;
   END_IF;
   IF NOT #DONE AND (#UNICODE = WCHAR#'ь') THEN
       #ASCII_HEX := 16#FC;
       #DONE := TRUE;
   END_IF;
   IF NOT #DONE AND (#UNICODE = WCHAR#'э') THEN
       #ASCII_HEX := 16#FD;
       #DONE := TRUE;
   END_IF;
END_REGION

REGION Network 23: ю | я |
   RUNG wire#powerrail
      I_Contact( #DONE )
      { S7_Templates := "SrcType := WChar" } EQ_Contact(in1 := #UNICODE, in2 := WCHAR#'ю')
      Move(in := 16#FE, out1 => #ASCII_HEX)
      S_Coil( #DONE )
   END_RUNG
   RUNG wire#powerrail
      I_Contact( #DONE )
      { S7_Templates := "SrcType := WChar" } EQ_Contact(in1 := #UNICODE, in2 := WCHAR#'я')
      Move(in := 16#FF, out1 => #ASCII_HEX)
      S_Coil( #DONE )
   END_RUNG
   // the same network as SCL:
   IF NOT #DONE AND (#UNICODE = WCHAR#'ю') THEN
       #ASCII_HEX := 16#FE;
       #DONE := TRUE;
   END_IF;
   IF NOT #DONE AND (#UNICODE = WCHAR#'я') THEN
       #ASCII_HEX := 16#FF;
       #DONE := TRUE;
   END_IF;
END_REGION

REGION Network 24: A | B | C | D | E |
   RUNG wire#powerrail
      I_Contact( #DONE )
      { S7_Templates := "SrcType := WChar" } EQ_Contact(in1 := #UNICODE, in2 := WCHAR#'A')
      Move(in := 16#41, out1 => #ASCII_HEX)
      S_Coil( #DONE )
   END_RUNG
   RUNG wire#powerrail
      I_Contact( #DONE )
      { S7_Templates := "SrcType := WChar" } EQ_Contact(in1 := #UNICODE, in2 := WCHAR#'B')
      Move(in := 16#42, out1 => #ASCII_HEX)
      S_Coil( #DONE )
   END_RUNG
   RUNG wire#powerrail
      I_Contact( #DONE )
      { S7_Templates := "SrcType := WChar" } EQ_Contact(in1 := #UNICODE, in2 := WCHAR#'C')
      Move(in := 16#43, out1 => #ASCII_HEX)
      S_Coil( #DONE )
   END_RUNG
   RUNG wire#powerrail
      I_Contact( #DONE )
      { S7_Templates := "SrcType := WChar" } EQ_Contact(in1 := #UNICODE, in2 := WCHAR#'D')
      Move(in := 16#44, out1 => #ASCII_HEX)
      S_Coil( #DONE )
   END_RUNG
   RUNG wire#powerrail
      I_Contact( #DONE )
      { S7_Templates := "SrcType := WChar" } EQ_Contact(in1 := #UNICODE, in2 := WCHAR#'E')
      Move(in := 16#45, out1 => #ASCII_HEX)
      S_Coil( #DONE )
   END_RUNG
   // the same network as SCL:
   IF NOT #DONE AND (#UNICODE = WCHAR#'A') THEN
       #ASCII_HEX := 16#41;
       #DONE := TRUE;
   END_IF;
   IF NOT #DONE AND (#UNICODE = WCHAR#'B') THEN
       #ASCII_HEX := 16#42;
       #DONE := TRUE;
   END_IF;
   IF NOT #DONE AND (#UNICODE = WCHAR#'C') THEN
       #ASCII_HEX := 16#43;
       #DONE := TRUE;
   END_IF;
   IF NOT #DONE AND (#UNICODE = WCHAR#'D') THEN
       #ASCII_HEX := 16#44;
       #DONE := TRUE;
   END_IF;
   IF NOT #DONE AND (#UNICODE = WCHAR#'E') THEN
       #ASCII_HEX := 16#45;
       #DONE := TRUE;
   END_IF;
END_REGION

REGION Network 25: F | G | H | I | J |
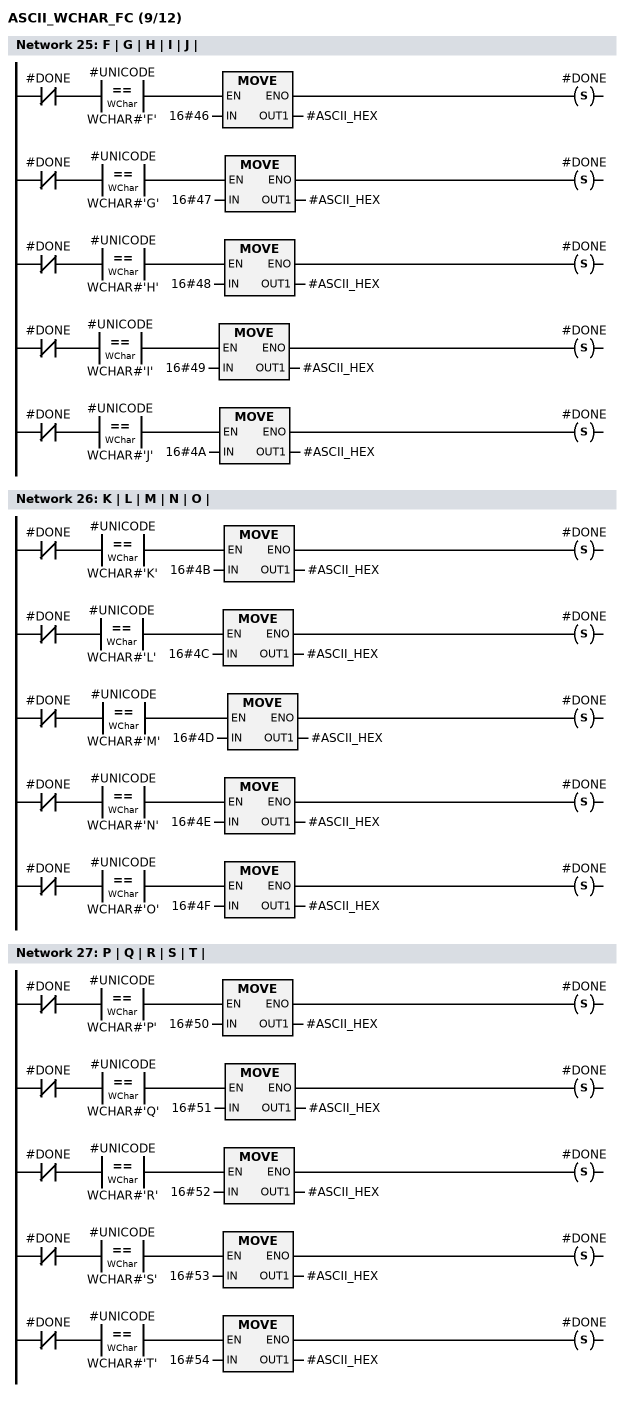
   RUNG wire#powerrail
      I_Contact( #DONE )
      { S7_Templates := "SrcType := WChar" } EQ_Contact(in1 := #UNICODE, in2 := WCHAR#'F')
      Move(in := 16#46, out1 => #ASCII_HEX)
      S_Coil( #DONE )
   END_RUNG
   RUNG wire#powerrail
      I_Contact( #DONE )
      { S7_Templates := "SrcType := WChar" } EQ_Contact(in1 := #UNICODE, in2 := WCHAR#'G')
      Move(in := 16#47, out1 => #ASCII_HEX)
      S_Coil( #DONE )
   END_RUNG
   RUNG wire#powerrail
      I_Contact( #DONE )
      { S7_Templates := "SrcType := WChar" } EQ_Contact(in1 := #UNICODE, in2 := WCHAR#'H')
      Move(in := 16#48, out1 => #ASCII_HEX)
      S_Coil( #DONE )
   END_RUNG
   RUNG wire#powerrail
      I_Contact( #DONE )
      { S7_Templates := "SrcType := WChar" } EQ_Contact(in1 := #UNICODE, in2 := WCHAR#'I')
      Move(in := 16#49, out1 => #ASCII_HEX)
      S_Coil( #DONE )
   END_RUNG
   RUNG wire#powerrail
      I_Contact( #DONE )
      { S7_Templates := "SrcType := WChar" } EQ_Contact(in1 := #UNICODE, in2 := WCHAR#'J')
      Move(in := 16#4A, out1 => #ASCII_HEX)
      S_Coil( #DONE )
   END_RUNG
   // the same network as SCL:
   IF NOT #DONE AND (#UNICODE = WCHAR#'F') THEN
       #ASCII_HEX := 16#46;
       #DONE := TRUE;
   END_IF;
   IF NOT #DONE AND (#UNICODE = WCHAR#'G') THEN
       #ASCII_HEX := 16#47;
       #DONE := TRUE;
   END_IF;
   IF NOT #DONE AND (#UNICODE = WCHAR#'H') THEN
       #ASCII_HEX := 16#48;
       #DONE := TRUE;
   END_IF;
   IF NOT #DONE AND (#UNICODE = WCHAR#'I') THEN
       #ASCII_HEX := 16#49;
       #DONE := TRUE;
   END_IF;
   IF NOT #DONE AND (#UNICODE = WCHAR#'J') THEN
       #ASCII_HEX := 16#4A;
       #DONE := TRUE;
   END_IF;
END_REGION

REGION Network 26: K | L | M | N | O |
   RUNG wire#powerrail
      I_Contact( #DONE )
      { S7_Templates := "SrcType := WChar" } EQ_Contact(in1 := #UNICODE, in2 := WCHAR#'K')
      Move(in := 16#4B, out1 => #ASCII_HEX)
      S_Coil( #DONE )
   END_RUNG
   RUNG wire#powerrail
      I_Contact( #DONE )
      { S7_Templates := "SrcType := WChar" } EQ_Contact(in1 := #UNICODE, in2 := WCHAR#'L')
      Move(in := 16#4C, out1 => #ASCII_HEX)
      S_Coil( #DONE )
   END_RUNG
   RUNG wire#powerrail
      I_Contact( #DONE )
      { S7_Templates := "SrcType := WChar" } EQ_Contact(in1 := #UNICODE, in2 := WCHAR#'M')
      Move(in := 16#4D, out1 => #ASCII_HEX)
      S_Coil( #DONE )
   END_RUNG
   RUNG wire#powerrail
      I_Contact( #DONE )
      { S7_Templates := "SrcType := WChar" } EQ_Contact(in1 := #UNICODE, in2 := WCHAR#'N')
      Move(in := 16#4E, out1 => #ASCII_HEX)
      S_Coil( #DONE )
   END_RUNG
   RUNG wire#powerrail
      I_Contact( #DONE )
      { S7_Templates := "SrcType := WChar" } EQ_Contact(in1 := #UNICODE, in2 := WCHAR#'O')
      Move(in := 16#4F, out1 => #ASCII_HEX)
      S_Coil( #DONE )
   END_RUNG
   // the same network as SCL:
   IF NOT #DONE AND (#UNICODE = WCHAR#'K') THEN
       #ASCII_HEX := 16#4B;
       #DONE := TRUE;
   END_IF;
   IF NOT #DONE AND (#UNICODE = WCHAR#'L') THEN
       #ASCII_HEX := 16#4C;
       #DONE := TRUE;
   END_IF;
   IF NOT #DONE AND (#UNICODE = WCHAR#'M') THEN
       #ASCII_HEX := 16#4D;
       #DONE := TRUE;
   END_IF;
   IF NOT #DONE AND (#UNICODE = WCHAR#'N') THEN
       #ASCII_HEX := 16#4E;
       #DONE := TRUE;
   END_IF;
   IF NOT #DONE AND (#UNICODE = WCHAR#'O') THEN
       #ASCII_HEX := 16#4F;
       #DONE := TRUE;
   END_IF;
END_REGION

REGION Network 27: P | Q | R | S | T |
   RUNG wire#powerrail
      I_Contact( #DONE )
      { S7_Templates := "SrcType := WChar" } EQ_Contact(in1 := #UNICODE, in2 := WCHAR#'P')
      Move(in := 16#50, out1 => #ASCII_HEX)
      S_Coil( #DONE )
   END_RUNG
   RUNG wire#powerrail
      I_Contact( #DONE )
      { S7_Templates := "SrcType := WChar" } EQ_Contact(in1 := #UNICODE, in2 := WCHAR#'Q')
      Move(in := 16#51, out1 => #ASCII_HEX)
      S_Coil( #DONE )
   END_RUNG
   RUNG wire#powerrail
      I_Contact( #DONE )
      { S7_Templates := "SrcType := WChar" } EQ_Contact(in1 := #UNICODE, in2 := WCHAR#'R')
      Move(in := 16#52, out1 => #ASCII_HEX)
      S_Coil( #DONE )
   END_RUNG
   RUNG wire#powerrail
      I_Contact( #DONE )
      { S7_Templates := "SrcType := WChar" } EQ_Contact(in1 := #UNICODE, in2 := WCHAR#'S')
      Move(in := 16#53, out1 => #ASCII_HEX)
      S_Coil( #DONE )
   END_RUNG
   RUNG wire#powerrail
      I_Contact( #DONE )
      { S7_Templates := "SrcType := WChar" } EQ_Contact(in1 := #UNICODE, in2 := WCHAR#'T')
      Move(in := 16#54, out1 => #ASCII_HEX)
      S_Coil( #DONE )
   END_RUNG
   // the same network as SCL:
   IF NOT #DONE AND (#UNICODE = WCHAR#'P') THEN
       #ASCII_HEX := 16#50;
       #DONE := TRUE;
   END_IF;
   IF NOT #DONE AND (#UNICODE = WCHAR#'Q') THEN
       #ASCII_HEX := 16#51;
       #DONE := TRUE;
   END_IF;
   IF NOT #DONE AND (#UNICODE = WCHAR#'R') THEN
       #ASCII_HEX := 16#52;
       #DONE := TRUE;
   END_IF;
   IF NOT #DONE AND (#UNICODE = WCHAR#'S') THEN
       #ASCII_HEX := 16#53;
       #DONE := TRUE;
   END_IF;
   IF NOT #DONE AND (#UNICODE = WCHAR#'T') THEN
       #ASCII_HEX := 16#54;
       #DONE := TRUE;
   END_IF;
END_REGION

REGION Network 28: U | V | W | X | Y | Z |
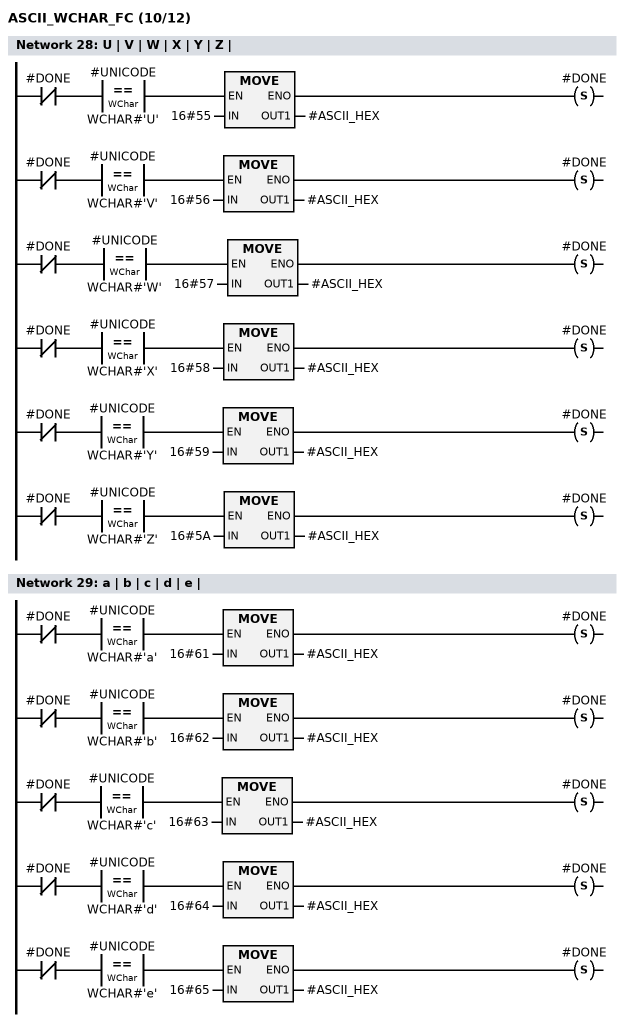
   RUNG wire#powerrail
      I_Contact( #DONE )
      { S7_Templates := "SrcType := WChar" } EQ_Contact(in1 := #UNICODE, in2 := WCHAR#'U')
      Move(in := 16#55, out1 => #ASCII_HEX)
      S_Coil( #DONE )
   END_RUNG
   RUNG wire#powerrail
      I_Contact( #DONE )
      { S7_Templates := "SrcType := WChar" } EQ_Contact(in1 := #UNICODE, in2 := WCHAR#'V')
      Move(in := 16#56, out1 => #ASCII_HEX)
      S_Coil( #DONE )
   END_RUNG
   RUNG wire#powerrail
      I_Contact( #DONE )
      { S7_Templates := "SrcType := WChar" } EQ_Contact(in1 := #UNICODE, in2 := WCHAR#'W')
      Move(in := 16#57, out1 => #ASCII_HEX)
      S_Coil( #DONE )
   END_RUNG
   RUNG wire#powerrail
      I_Contact( #DONE )
      { S7_Templates := "SrcType := WChar" } EQ_Contact(in1 := #UNICODE, in2 := WCHAR#'X')
      Move(in := 16#58, out1 => #ASCII_HEX)
      S_Coil( #DONE )
   END_RUNG
   RUNG wire#powerrail
      I_Contact( #DONE )
      { S7_Templates := "SrcType := WChar" } EQ_Contact(in1 := #UNICODE, in2 := WCHAR#'Y')
      Move(in := 16#59, out1 => #ASCII_HEX)
      S_Coil( #DONE )
   END_RUNG
   RUNG wire#powerrail
      I_Contact( #DONE )
      { S7_Templates := "SrcType := WChar" } EQ_Contact(in1 := #UNICODE, in2 := WCHAR#'Z')
      Move(in := 16#5A, out1 => #ASCII_HEX)
      S_Coil( #DONE )
   END_RUNG
   // the same network as SCL:
   IF NOT #DONE AND (#UNICODE = WCHAR#'U') THEN
       #ASCII_HEX := 16#55;
       #DONE := TRUE;
   END_IF;
   IF NOT #DONE AND (#UNICODE = WCHAR#'V') THEN
       #ASCII_HEX := 16#56;
       #DONE := TRUE;
   END_IF;
   IF NOT #DONE AND (#UNICODE = WCHAR#'W') THEN
       #ASCII_HEX := 16#57;
       #DONE := TRUE;
   END_IF;
   IF NOT #DONE AND (#UNICODE = WCHAR#'X') THEN
       #ASCII_HEX := 16#58;
       #DONE := TRUE;
   END_IF;
   IF NOT #DONE AND (#UNICODE = WCHAR#'Y') THEN
       #ASCII_HEX := 16#59;
       #DONE := TRUE;
   END_IF;
   IF NOT #DONE AND (#UNICODE = WCHAR#'Z') THEN
       #ASCII_HEX := 16#5A;
       #DONE := TRUE;
   END_IF;
END_REGION

REGION Network 29: a | b | c | d | e |
   RUNG wire#powerrail
      I_Contact( #DONE )
      { S7_Templates := "SrcType := WChar" } EQ_Contact(in1 := #UNICODE, in2 := WCHAR#'a')
      Move(in := 16#61, out1 => #ASCII_HEX)
      S_Coil( #DONE )
   END_RUNG
   RUNG wire#powerrail
      I_Contact( #DONE )
      { S7_Templates := "SrcType := WChar" } EQ_Contact(in1 := #UNICODE, in2 := WCHAR#'b')
      Move(in := 16#62, out1 => #ASCII_HEX)
      S_Coil( #DONE )
   END_RUNG
   RUNG wire#powerrail
      I_Contact( #DONE )
      { S7_Templates := "SrcType := WChar" } EQ_Contact(in1 := #UNICODE, in2 := WCHAR#'c')
      Move(in := 16#63, out1 => #ASCII_HEX)
      S_Coil( #DONE )
   END_RUNG
   RUNG wire#powerrail
      I_Contact( #DONE )
      { S7_Templates := "SrcType := WChar" } EQ_Contact(in1 := #UNICODE, in2 := WCHAR#'d')
      Move(in := 16#64, out1 => #ASCII_HEX)
      S_Coil( #DONE )
   END_RUNG
   RUNG wire#powerrail
      I_Contact( #DONE )
      { S7_Templates := "SrcType := WChar" } EQ_Contact(in1 := #UNICODE, in2 := WCHAR#'e')
      Move(in := 16#65, out1 => #ASCII_HEX)
      S_Coil( #DONE )
   END_RUNG
   // the same network as SCL:
   IF NOT #DONE AND (#UNICODE = WCHAR#'a') THEN
       #ASCII_HEX := 16#61;
       #DONE := TRUE;
   END_IF;
   IF NOT #DONE AND (#UNICODE = WCHAR#'b') THEN
       #ASCII_HEX := 16#62;
       #DONE := TRUE;
   END_IF;
   IF NOT #DONE AND (#UNICODE = WCHAR#'c') THEN
       #ASCII_HEX := 16#63;
       #DONE := TRUE;
   END_IF;
   IF NOT #DONE AND (#UNICODE = WCHAR#'d') THEN
       #ASCII_HEX := 16#64;
       #DONE := TRUE;
   END_IF;
   IF NOT #DONE AND (#UNICODE = WCHAR#'e') THEN
       #ASCII_HEX := 16#65;
       #DONE := TRUE;
   END_IF;
END_REGION

REGION Network 30: f | g | h | i | j |
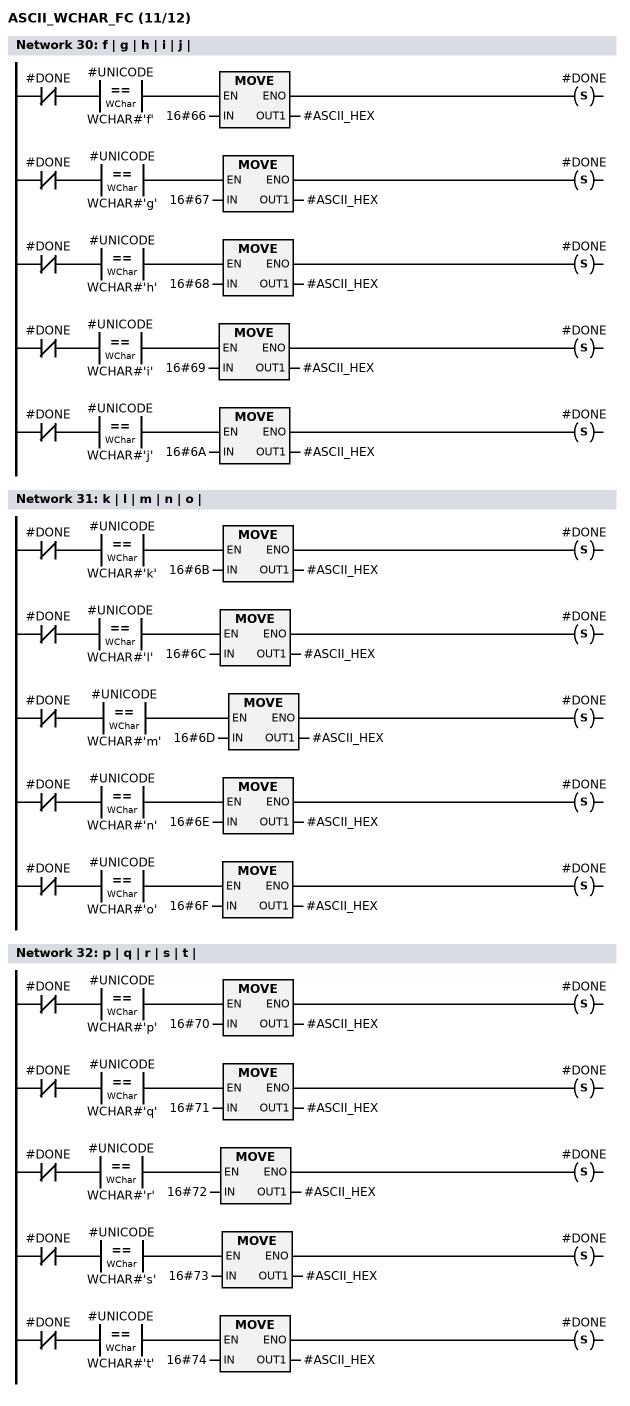
   RUNG wire#powerrail
      I_Contact( #DONE )
      { S7_Templates := "SrcType := WChar" } EQ_Contact(in1 := #UNICODE, in2 := WCHAR#'f')
      Move(in := 16#66, out1 => #ASCII_HEX)
      S_Coil( #DONE )
   END_RUNG
   RUNG wire#powerrail
      I_Contact( #DONE )
      { S7_Templates := "SrcType := WChar" } EQ_Contact(in1 := #UNICODE, in2 := WCHAR#'g')
      Move(in := 16#67, out1 => #ASCII_HEX)
      S_Coil( #DONE )
   END_RUNG
   RUNG wire#powerrail
      I_Contact( #DONE )
      { S7_Templates := "SrcType := WChar" } EQ_Contact(in1 := #UNICODE, in2 := WCHAR#'h')
      Move(in := 16#68, out1 => #ASCII_HEX)
      S_Coil( #DONE )
   END_RUNG
   RUNG wire#powerrail
      I_Contact( #DONE )
      { S7_Templates := "SrcType := WChar" } EQ_Contact(in1 := #UNICODE, in2 := WCHAR#'i')
      Move(in := 16#69, out1 => #ASCII_HEX)
      S_Coil( #DONE )
   END_RUNG
   RUNG wire#powerrail
      I_Contact( #DONE )
      { S7_Templates := "SrcType := WChar" } EQ_Contact(in1 := #UNICODE, in2 := WCHAR#'j')
      Move(in := 16#6A, out1 => #ASCII_HEX)
      S_Coil( #DONE )
   END_RUNG
   // the same network as SCL:
   IF NOT #DONE AND (#UNICODE = WCHAR#'f') THEN
       #ASCII_HEX := 16#66;
       #DONE := TRUE;
   END_IF;
   IF NOT #DONE AND (#UNICODE = WCHAR#'g') THEN
       #ASCII_HEX := 16#67;
       #DONE := TRUE;
   END_IF;
   IF NOT #DONE AND (#UNICODE = WCHAR#'h') THEN
       #ASCII_HEX := 16#68;
       #DONE := TRUE;
   END_IF;
   IF NOT #DONE AND (#UNICODE = WCHAR#'i') THEN
       #ASCII_HEX := 16#69;
       #DONE := TRUE;
   END_IF;
   IF NOT #DONE AND (#UNICODE = WCHAR#'j') THEN
       #ASCII_HEX := 16#6A;
       #DONE := TRUE;
   END_IF;
END_REGION

REGION Network 31: k | l | m | n | o |
   RUNG wire#powerrail
      I_Contact( #DONE )
      { S7_Templates := "SrcType := WChar" } EQ_Contact(in1 := #UNICODE, in2 := WCHAR#'k')
      Move(in := 16#6B, out1 => #ASCII_HEX)
      S_Coil( #DONE )
   END_RUNG
   RUNG wire#powerrail
      I_Contact( #DONE )
      { S7_Templates := "SrcType := WChar" } EQ_Contact(in1 := #UNICODE, in2 := WCHAR#'l')
      Move(in := 16#6C, out1 => #ASCII_HEX)
      S_Coil( #DONE )
   END_RUNG
   RUNG wire#powerrail
      I_Contact( #DONE )
      { S7_Templates := "SrcType := WChar" } EQ_Contact(in1 := #UNICODE, in2 := WCHAR#'m')
      Move(in := 16#6D, out1 => #ASCII_HEX)
      S_Coil( #DONE )
   END_RUNG
   RUNG wire#powerrail
      I_Contact( #DONE )
      { S7_Templates := "SrcType := WChar" } EQ_Contact(in1 := #UNICODE, in2 := WCHAR#'n')
      Move(in := 16#6E, out1 => #ASCII_HEX)
      S_Coil( #DONE )
   END_RUNG
   RUNG wire#powerrail
      I_Contact( #DONE )
      { S7_Templates := "SrcType := WChar" } EQ_Contact(in1 := #UNICODE, in2 := WCHAR#'o')
      Move(in := 16#6F, out1 => #ASCII_HEX)
      S_Coil( #DONE )
   END_RUNG
   // the same network as SCL:
   IF NOT #DONE AND (#UNICODE = WCHAR#'k') THEN
       #ASCII_HEX := 16#6B;
       #DONE := TRUE;
   END_IF;
   IF NOT #DONE AND (#UNICODE = WCHAR#'l') THEN
       #ASCII_HEX := 16#6C;
       #DONE := TRUE;
   END_IF;
   IF NOT #DONE AND (#UNICODE = WCHAR#'m') THEN
       #ASCII_HEX := 16#6D;
       #DONE := TRUE;
   END_IF;
   IF NOT #DONE AND (#UNICODE = WCHAR#'n') THEN
       #ASCII_HEX := 16#6E;
       #DONE := TRUE;
   END_IF;
   IF NOT #DONE AND (#UNICODE = WCHAR#'o') THEN
       #ASCII_HEX := 16#6F;
       #DONE := TRUE;
   END_IF;
END_REGION

REGION Network 32: p | q | r | s | t |
   RUNG wire#powerrail
      I_Contact( #DONE )
      { S7_Templates := "SrcType := WChar" } EQ_Contact(in1 := #UNICODE, in2 := WCHAR#'p')
      Move(in := 16#70, out1 => #ASCII_HEX)
      S_Coil( #DONE )
   END_RUNG
   RUNG wire#powerrail
      I_Contact( #DONE )
      { S7_Templates := "SrcType := WChar" } EQ_Contact(in1 := #UNICODE, in2 := WCHAR#'q')
      Move(in := 16#71, out1 => #ASCII_HEX)
      S_Coil( #DONE )
   END_RUNG
   RUNG wire#powerrail
      I_Contact( #DONE )
      { S7_Templates := "SrcType := WChar" } EQ_Contact(in1 := #UNICODE, in2 := WCHAR#'r')
      Move(in := 16#72, out1 => #ASCII_HEX)
      S_Coil( #DONE )
   END_RUNG
   RUNG wire#powerrail
      I_Contact( #DONE )
      { S7_Templates := "SrcType := WChar" } EQ_Contact(in1 := #UNICODE, in2 := WCHAR#'s')
      Move(in := 16#73, out1 => #ASCII_HEX)
      S_Coil( #DONE )
   END_RUNG
   RUNG wire#powerrail
      I_Contact( #DONE )
      { S7_Templates := "SrcType := WChar" } EQ_Contact(in1 := #UNICODE, in2 := WCHAR#'t')
      Move(in := 16#74, out1 => #ASCII_HEX)
      S_Coil( #DONE )
   END_RUNG
   // the same network as SCL:
   IF NOT #DONE AND (#UNICODE = WCHAR#'p') THEN
       #ASCII_HEX := 16#70;
       #DONE := TRUE;
   END_IF;
   IF NOT #DONE AND (#UNICODE = WCHAR#'q') THEN
       #ASCII_HEX := 16#71;
       #DONE := TRUE;
   END_IF;
   IF NOT #DONE AND (#UNICODE = WCHAR#'r') THEN
       #ASCII_HEX := 16#72;
       #DONE := TRUE;
   END_IF;
   IF NOT #DONE AND (#UNICODE = WCHAR#'s') THEN
       #ASCII_HEX := 16#73;
       #DONE := TRUE;
   END_IF;
   IF NOT #DONE AND (#UNICODE = WCHAR#'t') THEN
       #ASCII_HEX := 16#74;
       #DONE := TRUE;
   END_IF;
END_REGION

REGION Network 33: u | v | w | x | y | z |
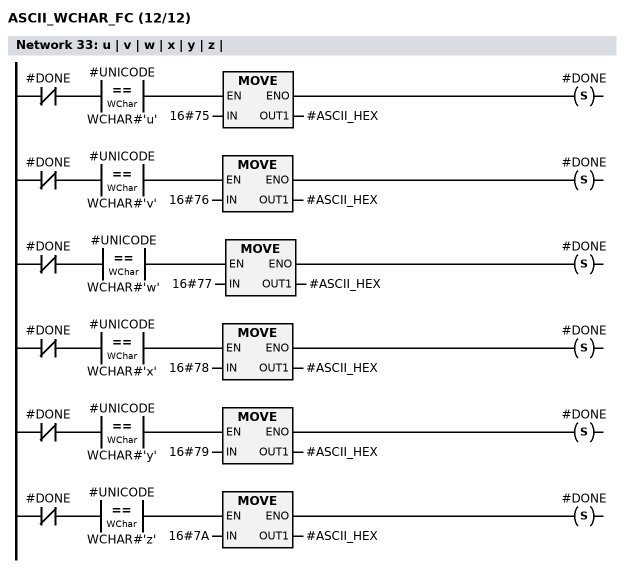
   RUNG wire#powerrail
      I_Contact( #DONE )
      { S7_Templates := "SrcType := WChar" } EQ_Contact(in1 := #UNICODE, in2 := WCHAR#'u')
      Move(in := 16#75, out1 => #ASCII_HEX)
      S_Coil( #DONE )
   END_RUNG
   RUNG wire#powerrail
      I_Contact( #DONE )
      { S7_Templates := "SrcType := WChar" } EQ_Contact(in1 := #UNICODE, in2 := WCHAR#'v')
      Move(in := 16#76, out1 => #ASCII_HEX)
      S_Coil( #DONE )
   END_RUNG
   RUNG wire#powerrail
      I_Contact( #DONE )
      { S7_Templates := "SrcType := WChar" } EQ_Contact(in1 := #UNICODE, in2 := WCHAR#'w')
      Move(in := 16#77, out1 => #ASCII_HEX)
      S_Coil( #DONE )
   END_RUNG
   RUNG wire#powerrail
      I_Contact( #DONE )
      { S7_Templates := "SrcType := WChar" } EQ_Contact(in1 := #UNICODE, in2 := WCHAR#'x')
      Move(in := 16#78, out1 => #ASCII_HEX)
      S_Coil( #DONE )
   END_RUNG
   RUNG wire#powerrail
      I_Contact( #DONE )
      { S7_Templates := "SrcType := WChar" } EQ_Contact(in1 := #UNICODE, in2 := WCHAR#'y')
      Move(in := 16#79, out1 => #ASCII_HEX)
      S_Coil( #DONE )
   END_RUNG
   RUNG wire#powerrail
      I_Contact( #DONE )
      { S7_Templates := "SrcType := WChar" } EQ_Contact(in1 := #UNICODE, in2 := WCHAR#'z')
      Move(in := 16#7A, out1 => #ASCII_HEX)
      S_Coil( #DONE )
   END_RUNG
   // the same network as SCL:
   IF NOT #DONE AND (#UNICODE = WCHAR#'u') THEN
       #ASCII_HEX := 16#75;
       #DONE := TRUE;
   END_IF;
   IF NOT #DONE AND (#UNICODE = WCHAR#'v') THEN
       #ASCII_HEX := 16#76;
       #DONE := TRUE;
   END_IF;
   IF NOT #DONE AND (#UNICODE = WCHAR#'w') THEN
       #ASCII_HEX := 16#77;
       #DONE := TRUE;
   END_IF;
   IF NOT #DONE AND (#UNICODE = WCHAR#'x') THEN
       #ASCII_HEX := 16#78;
       #DONE := TRUE;
   END_IF;
   IF NOT #DONE AND (#UNICODE = WCHAR#'y') THEN
       #ASCII_HEX := 16#79;
       #DONE := TRUE;
   END_IF;
   IF NOT #DONE AND (#UNICODE = WCHAR#'z') THEN
       #ASCII_HEX := 16#7A;
       #DONE := TRUE;
   END_IF;
END_REGION
END_FUNCTION

FUNCTION "ASCII_FC" : Void
{ S7_Optimized_Access := 'TRUE' }
VERSION : 0.1
   VAR_INPUT 
      Symbol : Char;
   END_VAR

   VAR_IN_OUT 
      Code : Byte;
      sys : Bool;
   END_VAR


BEGIN
	//числа от 0 до 9
	IF #sys = 0 THEN
	    IF #Symbol = '$00' THEN
	        #Code := 16#30;
	    END_IF;
	    IF #Symbol = '$01' THEN
	        #Code := 16#31;
	    END_IF;
	    IF #Symbol = '$02' THEN
	        #Code := 16#32;
	    END_IF;
	    IF #Symbol = '$03' THEN
	        #Code := 16#33;
	    END_IF;
	    IF #Symbol = '$04' THEN
	        #Code := 16#34;
	    END_IF;
	    IF #Symbol = '$05' THEN
	        #Code := 16#35;
	    END_IF;
	    IF #Symbol = '$06' THEN
	        #Code := 16#36;
	    END_IF;
	    IF #Symbol = '$07' THEN
	        #Code := 16#37;
	    END_IF;
	    IF #Symbol = '$08' THEN
	        #Code := 16#38;
	    END_IF;
	    IF #Symbol = '$09' THEN
	        #Code := 16#39;
	    END_IF;
	    IF #Symbol = '$0A' THEN
	        #Code := 16#41;
	    END_IF;
	    IF #Symbol = '$0B' THEN
	        #Code := 16#42;
	    END_IF;
	    IF #Symbol = '$0C' THEN
	        #Code := 16#43;
	    END_IF;
	    IF #Symbol = '$0D' THEN
	        #Code := 16#44;
	    END_IF;
	    IF #Symbol = '$0E' THEN
	        #Code := 16#45;
	    END_IF;
	    IF #Symbol = '$0F' THEN
	        #Code := 16#46;
	    END_IF;
	END_IF;
	
	//числа от 0 до 9
	IF #sys = 1 THEN
	    IF #Symbol = '$00' THEN
	        #Code := 16#30;
	    END_IF;
	    IF #Symbol = '$01' THEN
	        #Code := 16#31;
	    END_IF;
	    IF #Symbol = '$02' THEN
	        #Code := 16#32;
	    END_IF;
	    IF #Symbol = '$03' THEN
	        #Code := 16#33;
	    END_IF;
	    IF #Symbol = '$04' THEN
	        #Code := 16#34;
	    END_IF;
	    IF #Symbol = '$05' THEN
	        #Code := 16#35;
	    END_IF;
	    IF #Symbol = '$06' THEN
	        #Code := 16#36;
	    END_IF;
	    IF #Symbol = '$07' THEN
	        #Code := 16#37;
	    END_IF;
	    IF #Symbol = '$08' THEN
	        #Code := 16#38;
	    END_IF;
	    IF #Symbol = '$09' THEN
	        #Code := 16#39;
	    END_IF;
	    IF #Symbol = '$L' THEN
	        #Code := 16#41;
	    END_IF;
	    IF #Symbol = '$0B' THEN
	        #Code := 16#42;
	    END_IF;
	    IF #Symbol = '$P' THEN
	        #Code := 16#43;
	    END_IF;
	    IF #Symbol = '$R' THEN
	        #Code := 16#44;
	    END_IF;
	    IF #Symbol = '$0E' THEN
	        #Code := 16#45;
	    END_IF;
	    IF #Symbol = '$0F' THEN
	        #Code := 16#46;
	    END_IF;
	END_IF;
	
	
	
	//заглавные буквы А..Я
	
	
	//строчные буквы А..Я
	
	
	//специальные символы
	IF #Symbol = '?' THEN #Code := 16#3F; END_IF;
	IF #Symbol = '!' THEN #Code := 16#21; END_IF;
	IF #Symbol = '#' THEN #Code := 16#22; END_IF;
	
	//заглавные буквы A..Z
	IF #Symbol = 'g' THEN #Code := 16#67; END_IF;
	IF #Symbol = 'F' THEN #Code := 16#46; END_IF;
	//строчные буквы a..z
END_FUNCTION

FUNCTION "INT_TO_WSTRING" : Void
{ S7_Optimized_Access := 'TRUE' }
VERSION : 0.1
   VAR_INPUT 
      Value : Int;
      BASE : Array[0..9] of WChar;
      AsTime : Bool;
   END_VAR

   VAR_OUTPUT 
      "String" : WString;
   END_VAR

   VAR_TEMP 
      x1 : Int;
      x10 : Int;
      x100 : Int;
      x1000 : Int;
      x10000 : Int;
      "void" : WString[1];
   END_VAR


BEGIN
	#x10000 := #Value / 10000;
	#x1000 := (#Value - #x10000*10000) / 1000;
	#x100 := (#Value - #x10000*10000 - #x1000*1000) / 100;
	#x10 := (#Value - #x10000*10000- #x1000*1000 - #x100*100) / 10;
	#x1 := (#Value - #x10000 * 10000 - #x1000 * 1000 - #x100 * 100 - #x10 * 10) / 1;
	
	#String := #void;
	IF #x10000 > 0 THEN
	    #String := CONCAT_WSTRING(IN1 := #String, IN2 := #BASE[#x10000]);
	END_IF;
	
	IF #x1000 > 0 THEN
	    #String := CONCAT_WSTRING(IN1 := #String, IN2 := #BASE[#x1000]);
	ELSE
	    IF #x10000 > 0 THEN
	        #String := CONCAT_WSTRING(IN1 := #String, IN2 := #BASE[#x1000]);
	    END_IF;
	END_IF;
	
	IF #x100 > 0 THEN
	    #String := CONCAT_WSTRING(IN1 := #String, IN2 := #BASE[#x100]);
	ELSE
	    IF #x1000 > 0 OR #x10000 > 0 THEN
	        #String := CONCAT_WSTRING(IN1 := #String, IN2 := #BASE[#x100]);
	    END_IF;
	END_IF;
	
	IF #x10 > 0 THEN
	    #String := CONCAT_WSTRING(IN1 := #String, IN2 := #BASE[#x10]);
	ELSE
	    IF #x100 > 0 OR #x1000 > 0 OR #x10000 > 0 OR #AsTime THEN
	        #String := CONCAT_WSTRING(IN1 := #String, IN2 := #BASE[#x10]);
	    END_IF;
	END_IF;
	
	IF #x1 > 0 THEN
	    #String := CONCAT_WSTRING(IN1 := #String, IN2 := #BASE[#x1]);
	ELSE
	    IF #x10 > 0 OR #x100 > 0 OR #x1000 > 0 OR #x10000 > 0 OR #AsTime THEN
	        #String := CONCAT_WSTRING(IN1 := #String, IN2 := #BASE[#x1]);
	    END_IF;
	END_IF;
END_FUNCTION

DATA_BLOCK "ModBus_RTU_DB"   // DB30
VERSION : 0.1
// stored: AutoNumber false, DBAccessibleFromOPCUA true, InstanceOfName ModBus_RTU, InstanceOfType FB
"ModBus_RTU"
BEGIN
END_DATA_BLOCK

DATA_BLOCK "ModBus_TCP_DB"   // DB40
VERSION : 0.1
// stored: AutoNumber false, DBAccessibleFromOPCUA true, InstanceOfName ModBus_TCP, InstanceOfType FB
"ModBus_TCP"
BEGIN
   CONNECT.InterfaceId := 64;
   CONNECT.ID := 1;
   CONNECT.ConnectionType := 11;
   CONNECT.RemoteAddress.ADDR[1] := 192;
   CONNECT.RemoteAddress.ADDR[2] := 168;
   CONNECT.RemoteAddress.ADDR[3] := 0;
   CONNECT.RemoteAddress.ADDR[4] := 10;
   CONNECT.RemotePort := 502;
END_DATA_BLOCK

DATA_BLOCK "AIx_DB"   // DB220
VERSION : 0.1
// stored: AutoNumber false, DBAccessibleFromOPCUA true, InstanceOfName AIx, InstanceOfType FB
"AIx"
BEGIN
END_DATA_BLOCK

DATA_BLOCK "AOx_DB"   // DB230
VERSION : 0.1
// stored: AutoNumber false, DBAccessibleFromOPCUA true, InstanceOfName AOx, InstanceOfType FB
"AOx"
BEGIN
END_DATA_BLOCK

DATA_BLOCK "DIx_1_DB"   // DB200
VERSION : 0.1
// stored: AutoNumber false, DBAccessibleFromOPCUA true, InstanceOfName DIx_1, InstanceOfType FB
"DIx_1"
BEGIN
END_DATA_BLOCK

DATA_BLOCK "DOx_1_DB"   // DB210
VERSION : 0.1
// stored: AutoNumber false, DBAccessibleFromOPCUA true, InstanceOfName DOx_1, InstanceOfType FB
"DOx_1"
BEGIN
END_DATA_BLOCK

DATA_BLOCK "Motors_DB"   // DB240
VERSION : 0.1
// stored: AutoNumber false, DBAccessibleFromOPCUA true, InstanceOfName Motors, InstanceOfType FB
"Motors"
BEGIN
END_DATA_BLOCK

DATA_BLOCK "PIDx_DB"   // DB260
VERSION : 0.1
// stored: AutoNumber false, DBAccessibleFromOPCUA true, InstanceOfName PIDx, InstanceOfType FB
"PIDx"
BEGIN
END_DATA_BLOCK

DATA_BLOCK "Valves_DB"   // DB250
VERSION : 0.1
// stored: AutoNumber false, DBAccessibleFromOPCUA true, InstanceOfName Valves, InstanceOfType FB
"Valves"
BEGIN
END_DATA_BLOCK

DATA_BLOCK "FB_DRV_Start_DB"   // DB100
VERSION : 0.1
// stored: AutoNumber false, DBAccessibleFromOPCUA true, InstanceOfName FB_DRV_Start, InstanceOfType FB
"FB_DRV_Start"
BEGIN
END_DATA_BLOCK

DATA_BLOCK "Historian_DB"   // DB88
VERSION : 0.1
// stored: AutoNumber false, DBAccessibleFromOPCUA true, InstanceOfName Historian, InstanceOfType FB
"Historian"
BEGIN
END_DATA_BLOCK

DATA_BLOCK "Time_SYS_DB"   // DB95
VERSION : 0.1
// stored: AutoNumber false, DBAccessibleFromOPCUA true, InstanceOfName Time_SYS, InstanceOfType FB
"Time_SYS"
BEGIN
   TimeZone.Bias := 180;
   TimeZone.DaylightBias := 60;
   TimeZone.DaylightStartMonth := 3;
   TimeZone.DaylightStartWeek := 5;
   TimeZone.DaylightStartWeekday := 7;
   TimeZone.DaylightStartHour := 2;
   TimeZone.DaylightStartMinute := 0;
   TimeZone.StandardStartMonth := 10;
   TimeZone.StandardStartWeek := 5;
   TimeZone.StandardStartWeekday := 1;
   TimeZone.StandardStartHour := 3;
   TimeZone.StandardStartMinute := 0;
   TimeZone.TimeZoneName := 'GMT+3';
   SET_TIMEZONE.REQ := FALSE;
   SET_TIMEZONE.TimeZone.Bias := 180;
   SET_TIMEZONE.TimeZone.DaylightBias := 60;
   SET_TIMEZONE.TimeZone.DaylightStartMonth := 3;
   SET_TIMEZONE.TimeZone.DaylightStartWeek := 5;
   SET_TIMEZONE.TimeZone.DaylightStartWeekday := 7;
   SET_TIMEZONE.TimeZone.DaylightStartHour := 2;
   SET_TIMEZONE.TimeZone.DaylightStartMinute := 0;
   SET_TIMEZONE.TimeZone.StandardStartMonth := 10;
   SET_TIMEZONE.TimeZone.StandardStartWeek := 5;
   SET_TIMEZONE.TimeZone.StandardStartWeekday := 1;
   SET_TIMEZONE.TimeZone.StandardStartHour := 3;
   SET_TIMEZONE.TimeZone.StandardStartMinute := 0;
   SET_TIMEZONE.TimeZone.TimeZoneName := 'GMT+3';
   SET_TIMEZONE.DONE := FALSE;
   SET_TIMEZONE.BUSY := FALSE;
   SET_TIMEZONE.ERROR := FALSE;
   SET_TIMEZONE.STATUS := 16#7000;
END_DATA_BLOCK

DATA_BLOCK "AI_example_DB"   // DB300
VERSION : 0.1
// stored: AutoNumber false, DBAccessibleFromOPCUA true, InstanceOfName AI_ex, InstanceOfType FB
"AI_ex"
BEGIN
   Tx[0..1].SP := 3.0;
END_DATA_BLOCK

DATA_BLOCK "AO_example_DB"   // DB400
VERSION : 0.1
// stored: AutoNumber false, DBAccessibleFromOPCUA true, InstanceOfName AO_ex, InstanceOfType FB
"AO_ex"
BEGIN
END_DATA_BLOCK

DATA_BLOCK "M_DA_example_DB"   // DB600
VERSION : 0.1
// stored: AutoNumber false, DBAccessibleFromOPCUA true, InstanceOfName DRV_M_DA, InstanceOfType FB
"DRV_M_DA"
BEGIN
END_DATA_BLOCK

DATA_BLOCK "M_D_example_DB"   // DB500
VERSION : 0.1
// stored: AutoNumber false, DBAccessibleFromOPCUA true, InstanceOfName DRV_M_D, InstanceOfType FB
"DRV_M_D"
BEGIN
END_DATA_BLOCK

DATA_BLOCK "PID_example_DB"   // DB900
VERSION : 0.1
// stored: AutoNumber false, DBAccessibleFromOPCUA true, InstanceOfName PID_ex, InstanceOfType FB
"PID_ex"
BEGIN
END_DATA_BLOCK

DATA_BLOCK "V_D2A_example_DB"   // DB800
VERSION : 0.1
// stored: AutoNumber false, DBAccessibleFromOPCUA true, InstanceOfName DRV_V_D2A, InstanceOfType FB
"DRV_V_D2A"
BEGIN
END_DATA_BLOCK

DATA_BLOCK "V_D2_example_DB"   // DB700
VERSION : 0.1
// stored: AutoNumber false, DBAccessibleFromOPCUA true, InstanceOfName DRV_V_D2, InstanceOfType FB
"DRV_V_D2"
BEGIN
END_DATA_BLOCK

DATA_BLOCK "DB_Reset_All"   // DB1099
{ S7_Optimized_Access := 'TRUE' }
// stored: AutoNumber false, DBAccessibleFromOPCUA true, InstanceOfName IEC_TIMER, OfSystemLibElement IEC_TIMER, OfSystemLibVersion 1.0
"IEC_TIMER"
   // VAR
   //    PT : Time;
   //    ET { ExternalWritable := 'False'} : Time;
   //    IN : Bool;
   //    Q { ExternalWritable := 'False'} : Bool;
   // END_VAR
BEGIN
END_DATA_BLOCK

DATA_BLOCK "DB_pulse_01s"   // DB1100
{ S7_Optimized_Access := 'TRUE' }
// stored: AutoNumber false, DBAccessibleFromOPCUA true, InstanceOfName IEC_TIMER, OfSystemLibElement IEC_TIMER, OfSystemLibVersion 1.0
"IEC_TIMER"
   // VAR
   //    PT : Time;
   //    ET { ExternalWritable := 'False'} : Time;
   //    IN : Bool;
   //    Q { ExternalWritable := 'False'} : Bool;
   // END_VAR
BEGIN
END_DATA_BLOCK

DATA_BLOCK "DB_pulse_05s"   // DB1101
{ S7_Optimized_Access := 'TRUE' }
// stored: AutoNumber false, DBAccessibleFromOPCUA true, InstanceOfName IEC_TIMER, OfSystemLibElement IEC_TIMER, OfSystemLibVersion 1.0
"IEC_TIMER"
   // VAR
   //    PT : Time;
   //    ET { ExternalWritable := 'False'} : Time;
   //    IN : Bool;
   //    Q { ExternalWritable := 'False'} : Bool;
   // END_VAR
BEGIN
END_DATA_BLOCK

DATA_BLOCK "DB_pulse_10s"   // DB1104
{ S7_Optimized_Access := 'TRUE' }
// stored: AutoNumber false, DBAccessibleFromOPCUA true, InstanceOfName IEC_TIMER, OfSystemLibElement IEC_TIMER, OfSystemLibVersion 1.0
"IEC_TIMER"
   // VAR
   //    PT : Time;
   //    ET { ExternalWritable := 'False'} : Time;
   //    IN : Bool;
   //    Q { ExternalWritable := 'False'} : Bool;
   // END_VAR
BEGIN
END_DATA_BLOCK

DATA_BLOCK "DB_pulse_1m"   // DB1106
{ S7_Optimized_Access := 'TRUE' }
// stored: AutoNumber false, DBAccessibleFromOPCUA true, InstanceOfName IEC_TIMER, OfSystemLibElement IEC_TIMER, OfSystemLibVersion 1.0
"IEC_TIMER"
   // VAR
   //    PT : Time;
   //    ET { ExternalWritable := 'False'} : Time;
   //    IN : Bool;
   //    Q { ExternalWritable := 'False'} : Bool;
   // END_VAR
BEGIN
END_DATA_BLOCK

DATA_BLOCK "DB_pulse_1s"   // DB1102
{ S7_Optimized_Access := 'TRUE' }
// stored: AutoNumber false, DBAccessibleFromOPCUA true, InstanceOfName IEC_TIMER, OfSystemLibElement IEC_TIMER, OfSystemLibVersion 1.0
"IEC_TIMER"
   // VAR
   //    PT : Time;
   //    ET { ExternalWritable := 'False'} : Time;
   //    IN : Bool;
   //    Q { ExternalWritable := 'False'} : Bool;
   // END_VAR
BEGIN
END_DATA_BLOCK

DATA_BLOCK "DB_pulse_30s"   // DB1105
{ S7_Optimized_Access := 'TRUE' }
// stored: AutoNumber false, DBAccessibleFromOPCUA true, InstanceOfName IEC_TIMER, OfSystemLibElement IEC_TIMER, OfSystemLibVersion 1.0
"IEC_TIMER"
   // VAR
   //    PT : Time;
   //    ET { ExternalWritable := 'False'} : Time;
   //    IN : Bool;
   //    Q { ExternalWritable := 'False'} : Bool;
   // END_VAR
BEGIN
END_DATA_BLOCK

DATA_BLOCK "DB_pulse_5s"   // DB1103
{ S7_Optimized_Access := 'TRUE' }
// stored: AutoNumber false, DBAccessibleFromOPCUA true, InstanceOfName IEC_TIMER, OfSystemLibElement IEC_TIMER, OfSystemLibVersion 1.0
"IEC_TIMER"
   // VAR
   //    PT : Time;
   //    ET { ExternalWritable := 'False'} : Time;
   //    IN : Bool;
   //    Q { ExternalWritable := 'False'} : Bool;
   // END_VAR
BEGIN
END_DATA_BLOCK
